LIN {X 0,Y 533.532,Z 613.937,A -85,B 0,C 180,E1 -4225.939,E2 -4225.939} C_VEL
LIN {X 0,Y 532.908,Z 627.148,A -85,B 0,C 180,E1 -4226.975,E2 -4226.975} C_VEL
LIN {X 0,Y 532.504,Z 637.558,A -85,B 0,C 180,E1 -4227.919,E2 -4227.919} C_VEL
LIN {X 0,Y 532.126,Z 646.759,A -85,B 0,C 180,E1 -4228.864,E2 -4228.864} C_VEL
LIN {X 0,Y 531.704,Z 656.519,A -85,B 0,C 180,E1 -4229.999,E2 -4229.999} C_VEL
LIN {X 0,Y 531.313,Z 666.406,A -85,B 0,C 180,E1 -4231.326,E2 -4231.326} C_VEL
LIN {X 0,Y 531.018,Z 676.107,A -85,B 0,C 180,E1 -4232.844,E2 -4232.844} C_VEL
LIN {X 0,Y 530.774,Z 685.128,A -85,B 0,C 180,E1 -4234.556,E2 -4234.556} C_VEL
LIN {X 0,Y 530.628,Z 691.8,A -85,B 0,C 180,E1 -4236.081,E2 -4236.081} C_VEL
LIN {X 0,Y 530.552,Z 697.288,A -85,B 0,C 180,E1 -4237.611,E2 -4237.611} C_VEL
LIN {X 0,Y 530.429,Z 701.704,A -85,B 0,C 180,E1 -4239.148,E2 -4239.148} C_VEL
LIN {X 0,Y 530.423,Z 705.038,A -85,B 0,C 180,E1 -4240.689,E2 -4240.689} C_VEL
LIN {X 0,Y 530.38,Z 707.363,A -85,B 0,C 180,E1 -4242.239,E2 -4242.239} C_VEL
LIN {X 0,Y 530.39,Z 708.671,A -85,B 0,C 180,E1 -4243.798,E2 -4243.798} C_VEL
LIN {X 0,Y 530.314,Z 708.94,A -85,B 0,C 180,E1 -4245.369,E2 -4245.369} C_VEL
LIN {X 0,Y 530.358,Z 708.205,A -85,B 0,C 180,E1 -4246.949,E2 -4246.949} C_VEL
LIN {X 0,Y 530.365,Z 706.395,A -85,B 0,C 180,E1 -4248.543,E2 -4248.543} C_VEL
LIN {X 0,Y 530.391,Z 703.522,A -85,B 0,C 180,E1 -4250.151,E2 -4250.151} C_VEL
LIN {X 0,Y 530.516,Z 698.892,A -85,B 0,C 180,E1 -4251.978,E2 -4251.978} C_VEL
LIN {X 0,Y 530.594,Z 693.091,A -85,B 0,C 180,E1 -4253.684,E2 -4253.684} C_VEL
LIN {X 0,Y 530.727,Z 687.292,A -85,B 0,C 180,E1 -4255.07,E2 -4255.07} C_VEL
LIN {X 0,Y 530.922,Z 680.034,A -85,B 0,C 180,E1 -4256.535,E2 -4256.535} C_VEL
LIN {X 0,Y 531.158,Z 671.391,A -85,B 0,C 180,E1 -4258.015,E2 -4258.015} C_VEL
LIN {X 0,Y 531.539,Z 661.138,A -85,B 0,C 180,E1 -4259.505,E2 -4259.505} C_VEL
LIN {X 0,Y 531.98,Z 650.38,A -85,B 0,C 180,E1 -4260.826,E2 -4260.826} C_VEL
LIN {X 0,Y 532.443,Z 639.033,A -85,B 0,C 180,E1 -4262.027,E2 -4262.027} C_VEL
LIN {X 0,Y 532.896,Z 627.678,A -85,B 0,C 180,E1 -4263.069,E2 -4263.069} C_VEL
LIN {X 0,Y 533.43,Z 615.355,A -85,B 0,C 180,E1 -4264.046,E2 -4264.046} C_VEL
LIN {X 0,Y 534.028,Z 600.641,A -85,B 0,C 180,E1 -4265.037,E2 -4265.037} C_VEL
LIN {X 0,Y 534.612,Z 585.573,A -85,B 0,C 180,E1 -4265.859,E2 -4265.859} C_VEL
LIN {X 0,Y 535.013,Z 571.807,A -85,B 0,C 180,E1 -4266.478,E2 -4266.478} C_VEL
LIN {X 0,Y 535.43,Z 558.758,A -85,B 0,C 180,E1 -4266.948,E2 -4266.948} C_VEL
LIN {X 0,Y 535.723,Z 546.011,A -85,B 0,C 180,E1 -4267.312,E2 -4267.312} C_VEL
LIN {X 0,Y 535.688,Z 538.488,A -85,B 0,C 180,E1 -4267.498,E2 -4267.498} C_VEL
LIN {X 0,Y 530.646,Z 521.655,A -85,B 0,C 180,E1 -4268.016,E2 -4268.016} C_VEL
LIN {X 0,Y 530.688,Z 516.304,A -85,B 0,C 180,E1 -4270.986,E2 -4270.986} C_VEL
LIN {X 0,Y 530.788,Z 512.053,A -85,B 0,C 180,E1 -4273.511,E2 -4273.511} C_VEL
LIN {X 0,Y 530.883,Z 506.871,A -85,B 0,C 180,E1 -4276.496,E2 -4276.496} C_VEL
LIN {X 0,Y 530.93,Z 502.507,A -85,B 0,C 180,E1 -4278.981,E2 -4278.981} C_VEL
LIN {X 0,Y 530.941,Z 497.816,A -85,B 0,C 180,E1 -4281.527,E2 -4281.527} C_VEL
LIN {X 0,Y 531.038,Z 492.653,A -85,B 0,C 180,E1 -4284.288,E2 -4284.288} C_VEL
LIN {X 0,Y 530.968,Z 492.661,A -85,B 0,C 180,E1 -4287.133,E2 -4287.133} C_VEL
LIN {X 0,Y 530.979,Z 492.659,A -85,B 0,C 180,E1 -4289.803,E2 -4289.803} C_VEL
LIN {X 0,Y 531.01,Z 492.655,A -85,B 0,C 180,E1 -4292.465,E2 -4292.465} C_VEL
LIN {X 0,Y 531.007,Z 492.656,A -85,B 0,C 180,E1 -4294.942,E2 -4294.942} C_VEL
LIN {X 0,Y 530.983,Z 492.658,A -85,B 0,C 180,E1 -4297.893,E2 -4297.893} C_VEL
LIN {X 0,Y 530.989,Z 492.655,A -85,B 0,C 180,E1 -4300.677,E2 -4300.677} C_VEL
LIN {X 0,Y 530.984,Z 492.658,A -85,B 0,C 180,E1 -4303.071,E2 -4303.071} C_VEL
LIN {X 0,Y 531.009,Z 492.654,A -85,B 0,C 180,E1 -4305.435,E2 -4305.435} C_VEL
LIN {X 0,Y 531.037,Z 492.65,A -85,B 0,C 180,E1 -4308.549,E2 -4308.549} C_VEL
LIN {X 0,Y 531.051,Z 492.646,A -85,B 0,C 180,E1 -4311.629,E2 -4311.629} C_VEL
LIN {X 0,Y 531.137,Z 492.636,A -85,B 0,C 180,E1 -4314.685,E2 -4314.685} C_VEL
LIN {X 0,Y 531.134,Z 492.639,A -85,B 0,C 180,E1 -4317.725,E2 -4317.725} C_VEL
LIN {X 0,Y 531.147,Z 492.638,A -85,B 0,C 180,E1 -4320.758,E2 -4320.758} C_VEL
LIN {X 0,Y 531.101,Z 492.641,A -85,B 0,C 180,E1 -4323.034,E2 -4323.034} C_VEL
LIN {X 0,Y 531.074,Z 492.645,A -85,B 0,C 180,E1 -4326.077,E2 -4326.077} C_VEL
LIN {X 0,Y 531.026,Z 492.65,A -85,B 0,C 180,E1 -4329.138,E2 -4329.138} C_VEL
LIN {X 0,Y 531.03,Z 492.647,A -85,B 0,C 180,E1 -4332.225,E2 -4332.225} C_VEL
LIN {X 0,Y 530.985,Z 492.656,A -85,B 0,C 180,E1 -4335.35,E2 -4335.35} C_VEL
LIN {X 0,Y 531.005,Z 492.639,A -85,B 0,C 180,E1 -4337.722,E2 -4337.722} C_VEL
LIN {X 0,Y 530.994,Z 492.657,A -85,B 0,C 180,E1 -4340.938,E2 -4340.938} C_VEL
LIN {X 0,Y 530.997,Z 492.644,A -85,B 0,C 180,E1 -4344.045,E2 -4344.045} C_VEL
LIN {X 0,Y 531.002,Z 492.655,A -85,B 0,C 180,E1 -4346.743,E2 -4346.743} C_VEL
LIN {X 0,Y 530.99,Z 492.658,A -85,B 0,C 180,E1 -4349.322,E2 -4349.322} C_VEL
LIN {X 0,Y 530.97,Z 492.66,A -85,B 0,C 180,E1 -4352.104,E2 -4352.104} C_VEL
LIN {X 0,Y 530.982,Z 492.657,A -85,B 0,C 180,E1 -4354.855,E2 -4354.855} C_VEL
LIN {X 0,Y 530.964,Z 492.66,A -85,B 0,C 180,E1 -4357.507,E2 -4357.507} C_VEL
LIN {X 0,Y 531.019,Z 492.652,A -85,B 0,C 180,E1 -4360.429,E2 -4360.429} C_VEL
LIN {X 0,Y 530.957,Z 492.661,A -85,B 0,C 180,E1 -4363.495,E2 -4363.495} C_VEL
LIN {X 0,Y 531.009,Z 492.819,A -85,B 0,C 180,E1 -4366.402,E2 -4366.402} C_VEL
LIN {X 0,Y 532.868,Z 501.243,A -85,B 0,C 180,E1 -4368.744,E2 -4368.744} C_VEL
LIN {X 0,Y 533.677,Z 505.22,A -85,B 0,C 180,E1 -4369.815,E2 -4369.815} C_VEL
LIN {X 0,Y 533.689,Z 513.013,A -85,B 0,C 180,E1 -4371.764,E2 -4371.764} C_VEL
LIN {X 0,Y 533.387,Z 525.433,A -85,B 0,C 180,E1 -4374.777,E2 -4374.777} C_VEL
LIN {X 0,Y 532.901,Z 537.907,A -85,B 0,C 180,E1 -4377.86,E2 -4377.86} C_VEL
LIN {X 0,Y 532.51,Z 550.04,A -85,B 0,C 180,E1 -4380.771,E2 -4380.771} C_VEL
LIN {X 0,Y 532.194,Z 560.938,A -85,B 0,C 180,E1 -4383.322,E2 -4383.322} C_VEL
LIN {X 0,Y 531.825,Z 573.652,A -85,B 0,C 180,E1 -4386.232,E2 -4386.232} C_VEL
LIN {X 0,Y 531.761,Z 577.116,A -85,B 0,C 180,E1 -4387.016,E2 -4387.016} C_VEL
LIN {X 0,Y 535.893,Z 592.599,A -85,B 0,C 180,E1 -4387.446,E2 -4387.446} C_VEL
LIN {X 0,Y 535.686,Z 608.888,A -85,B 0,C 180,E1 -4387.805,E2 -4387.805} C_VEL
LIN {X 0,Y 535.309,Z 624.847,A -85,B 0,C 180,E1 -4388.3,E2 -4388.3} C_VEL
LIN {X 0,Y 534.788,Z 640.031,A -85,B 0,C 180,E1 -4388.916,E2 -4388.916} C_VEL
LIN {X 0,Y 534.26,Z 655.297,A -85,B 0,C 180,E1 -4389.7,E2 -4389.7} C_VEL
LIN {X 0,Y 533.646,Z 670.869,A -85,B 0,C 180,E1 -4390.678,E2 -4390.678} C_VEL
LIN {X 0,Y 533.025,Z 685.379,A -85,B 0,C 180,E1 -4391.779,E2 -4391.779} C_VEL
LIN {X 0,Y 532.488,Z 698.13,A -85,B 0,C 180,E1 -4392.924,E2 -4392.924} C_VEL
LIN {X 0,Y 532.031,Z 709.292,A -85,B 0,C 180,E1 -4394.093,E2 -4394.093} C_VEL
LIN {X 0,Y 531.635,Z 720.431,A -85,B 0,C 180,E1 -4395.454,E2 -4395.454} C_VEL
LIN {X 0,Y 531.191,Z 731.218,A -85,B 0,C 180,E1 -4397.003,E2 -4397.003} C_VEL
LIN {X 0,Y 530.965,Z 740.269,A -85,B 0,C 180,E1 -4398.549,E2 -4398.549} C_VEL
LIN {X 0,Y 530.696,Z 747.861,A -85,B 0,C 180,E1 -4400.088,E2 -4400.088} C_VEL
LIN {X 0,Y 530.568,Z 755.47,A -85,B 0,C 180,E1 -4402.006,E2 -4402.006} C_VEL
LIN {X 0,Y 530.494,Z 761.25,A -85,B 0,C 180,E1 -4403.917,E2 -4403.917} C_VEL
LIN {X 0,Y 530.403,Z 764.638,A -85,B 0,C 180,E1 -4405.441,E2 -4405.441} C_VEL
LIN {X 0,Y 530.444,Z 767.09,A -85,B 0,C 180,E1 -4406.963,E2 -4406.963} C_VEL
LIN {X 0,Y 530.357,Z 768.48,A -85,B 0,C 180,E1 -4408.482,E2 -4408.482} C_VEL
LIN {X 0,Y 530.338,Z 769,A -85,B 0,C 180,E1 -4410.001,E2 -4410.001} C_VEL
LIN {X 0,Y 530.357,Z 768.479,A -85,B 0,C 180,E1 -4411.519,E2 -4411.519} C_VEL
LIN {X 0,Y 530.444,Z 767.087,A -85,B 0,C 180,E1 -4413.039,E2 -4413.039} C_VEL
LIN {X 0,Y 530.404,Z 764.635,A -85,B 0,C 180,E1 -4414.561,E2 -4414.561} C_VEL
LIN {X 0,Y 530.494,Z 761.247,A -85,B 0,C 180,E1 -4416.085,E2 -4416.085} C_VEL
LIN {X 0,Y 530.57,Z 755.465,A -85,B 0,C 180,E1 -4417.996,E2 -4417.996} C_VEL
LIN {X 0,Y 530.697,Z 747.853,A -85,B 0,C 180,E1 -4419.914,E2 -4419.914} C_VEL
LIN {X 0,Y 531.001,Z 739.244,A -85,B 0,C 180,E1 -4421.646,E2 -4421.646} C_VEL
LIN {X 0,Y 531.229,Z 729.97,A -85,B 0,C 180,E1 -4423.193,E2 -4423.193} C_VEL
LIN {X 0,Y 531.68,Z 719.216,A -85,B 0,C 180,E1 -4424.704,E2 -4424.704} C_VEL
LIN {X 0,Y 532.103,Z 707.5,A -85,B 0,C 180,E1 -4426.104,E2 -4426.104} C_VEL
LIN {X 0,Y 532.631,Z 695.034,A -85,B 0,C 180,E1 -4427.37,E2 -4427.37} C_VEL
LIN {X 0,Y 533.201,Z 681.455,A -85,B 0,C 180,E1 -4428.542,E2 -4428.542} C_VEL
LIN {X 0,Y 533.812,Z 666.56,A -85,B 0,C 180,E1 -4429.617,E2 -4429.617} C_VEL
LIN {X 0,Y 534.389,Z 651.742,A -85,B 0,C 180,E1 -4430.498,E2 -4430.498} C_VEL
LIN {X 0,Y 534.889,Z 637.688,A -85,B 0,C 180,E1 -4431.185,E2 -4431.185} C_VEL
LIN {X 0,Y 535.393,Z 622.424,A -85,B 0,C 180,E1 -4431.787,E2 -4431.787} C_VEL
LIN {X 0,Y 535.698,Z 606.492,A -85,B 0,C 180,E1 -4432.261,E2 -4432.261} C_VEL
LIN {X 0,Y 535.767,Z 592.182,A -85,B 0,C 180,E1 -4432.567,E2 -4432.567} C_VEL
LIN {X 0,Y 531.754,Z 577.091,A -85,B 0,C 180,E1 -4432.99,E2 -4432.99} C_VEL
LIN {X 0,Y 532.176,Z 562.417,A -85,B 0,C 180,E1 -4436.335,E2 -4436.335} C_VEL
LIN {X 0,Y 532.517,Z 550.032,A -85,B 0,C 180,E1 -4439.23,E2 -4439.23} C_VEL
LIN {X 0,Y 532.907,Z 537.9,A -85,B 0,C 180,E1 -4442.142,E2 -4442.142} C_VEL
LIN {X 0,Y 533.437,Z 524.602,A -85,B 0,C 180,E1 -4445.43,E2 -4445.43} C_VEL
LIN {X 0,Y 533.404,Z 512.664,A -85,B 0,C 180,E1 -4447.973,E2 -4447.973} C_VEL
LIN {X 0,Y 533.144,Z 503.532,A -85,B 0,C 180,E1 -4449.886,E2 -4449.886} C_VEL
LIN {X 0,Y 530.993,Z 492.658,A -85,B 0,C 180,E1 -4452.38,E2 -4452.38} C_VEL
LIN {X 0,Y 530.989,Z 492.654,A -85,B 0,C 180,E1 -4455.621,E2 -4455.621} C_VEL
LIN {X 0,Y 530.997,Z 492.658,A -85,B 0,C 180,E1 -4458.565,E2 -4458.565} C_VEL
LIN {X 0,Y 530.96,Z 492.657,A -85,B 0,C 180,E1 -4461.53,E2 -4461.53} C_VEL
LIN {X 0,Y 530.978,Z 492.661,A -85,B 0,C 180,E1 -4464.382,E2 -4464.382} C_VEL
LIN {X 0,Y 530.971,Z 492.656,A -85,B 0,C 180,E1 -4467.134,E2 -4467.134} C_VEL
LIN {X 0,Y 530.971,Z 492.659,A -85,B 0,C 180,E1 -4469.803,E2 -4469.803} C_VEL
LIN {X 0,Y 531.018,Z 492.653,A -85,B 0,C 180,E1 -4472.467,E2 -4472.467} C_VEL
LIN {X 0,Y 531.008,Z 492.651,A -85,B 0,C 180,E1 -4474.943,E2 -4474.943} C_VEL
LIN {X 0,Y 530.972,Z 492.658,A -85,B 0,C 180,E1 -4477.265,E2 -4477.265} C_VEL
LIN {X 0,Y 532.385,Z 496.563,A -85,B 0,C 180,E1 -4477.408,E2 -4477.408} C_VEL
LIN {X 0,Y 535.775,Z 504.819,A -85,B 0,C 180,E1 -4477.744,E2 -4477.744} C_VEL
LIN {X 0,Y 535.408,Z 520.411,A -85,B 0,C 180,E1 -4478.188,E2 -4478.188} C_VEL
LIN {X 0,Y 534.945,Z 536.534,A -85,B 0,C 180,E1 -4478.808,E2 -4478.808} C_VEL
LIN {X 0,Y 534.336,Z 552.771,A -85,B 0,C 180,E1 -4479.602,E2 -4479.602} C_VEL
LIN {X 0,Y 533.789,Z 567.376,A -85,B 0,C 180,E1 -4480.483,E2 -4480.483} C_VEL
LIN {X 0,Y 533.198,Z 582.144,A -85,B 0,C 180,E1 -4481.559,E2 -4481.559} C_VEL
LIN {X 0,Y 532.638,Z 595.622,A -85,B 0,C 180,E1 -4482.73,E2 -4482.73} C_VEL
LIN {X 0,Y 532.104,Z 607.116,A -85,B 0,C 180,E1 -4483.897,E2 -4483.897} C_VEL
LIN {X 0,Y 531.704,Z 618.906,A -85,B 0,C 180,E1 -4485.297,E2 -4485.297} C_VEL
LIN {X 0,Y 531.229,Z 629.714,A -85,B 0,C 180,E1 -4486.808,E2 -4486.808} C_VEL
LIN {X 0,Y 531.003,Z 638.994,A -85,B 0,C 180,E1 -4488.355,E2 -4488.355} C_VEL
LIN {X 0,Y 530.699,Z 647.635,A -85,B 0,C 180,E1 -4490.087,E2 -4490.087} C_VEL
LIN {X 0,Y 530.604,Z 653.896,A -85,B 0,C 180,E1 -4491.623,E2 -4491.623} C_VEL
LIN {X 0,Y 530.549,Z 658.995,A -85,B 0,C 180,E1 -4493.153,E2 -4493.153} C_VEL
LIN {X 0,Y 530.472,Z 662.97,A -85,B 0,C 180,E1 -4494.679,E2 -4494.679} C_VEL
LIN {X 0,Y 530.478,Z 665.916,A -85,B 0,C 180,E1 -4496.202,E2 -4496.202} C_VEL
LIN {X 0,Y 530.403,Z 667.872,A -85,B 0,C 180,E1 -4497.722,E2 -4497.722} C_VEL
LIN {X 0,Y 530.342,Z 668.857,A -85,B 0,C 180,E1 -4499.241,E2 -4499.241} C_VEL
LIN {X 0,Y 530.341,Z 668.874,A -85,B 0,C 180,E1 -4500.76,E2 -4500.76} C_VEL
LIN {X 0,Y 530.403,Z 667.951,A -85,B 0,C 180,E1 -4502.279,E2 -4502.279} C_VEL
LIN {X 0,Y 530.48,Z 666.057,A -85,B 0,C 180,E1 -4503.799,E2 -4503.799} C_VEL
LIN {X 0,Y 530.472,Z 663.168,A -85,B 0,C 180,E1 -4505.322,E2 -4505.322} C_VEL
LIN {X 0,Y 530.55,Z 659.27,A -85,B 0,C 180,E1 -4506.847,E2 -4506.847} C_VEL
LIN {X 0,Y 530.604,Z 654.24,A -85,B 0,C 180,E1 -4508.378,E2 -4508.378} C_VEL
LIN {X 0,Y 530.695,Z 648.056,A -85,B 0,C 180,E1 -4509.914,E2 -4509.914} C_VEL
LIN {X 0,Y 530.977,Z 639.556,A -85,B 0,C 180,E1 -4511.632,E2 -4511.632} C_VEL
LIN {X 0,Y 531.226,Z 630.266,A -85,B 0,C 180,E1 -4513.192,E2 -4513.192} C_VEL
LIN {X 0,Y 531.675,Z 619.59,A -85,B 0,C 180,E1 -4514.704,E2 -4514.704} C_VEL
LIN {X 0,Y 532.077,Z 607.953,A -85,B 0,C 180,E1 -4516.104,E2 -4516.104} C_VEL
LIN {X 0,Y 532.598,Z 595.538,A -85,B 0,C 180,E1 -4517.371,E2 -4517.371} C_VEL
LIN {X 0,Y 533.19,Z 582,A -85,B 0,C 180,E1 -4518.542,E2 -4518.542} C_VEL
LIN {X 0,Y 533.804,Z 567.184,A -85,B 0,C 180,E1 -4519.617,E2 -4519.617} C_VEL
LIN {X 0,Y 534.384,Z 552.56,A -85,B 0,C 180,E1 -4520.498,E2 -4520.498} C_VEL
LIN {X 0,Y 534.932,Z 537.448,A -85,B 0,C 180,E1 -4521.243,E2 -4521.243} C_VEL
LIN {X 0,Y 535.376,Z 520.293,A -85,B 0,C 180,E1 -4521.901,E2 -4521.901} C_VEL
LIN {X 0,Y 535.732,Z 506.697,A -85,B 0,C 180,E1 -4522.294,E2 -4522.294} C_VEL
LIN {X 0,Y 535.554,Z 504.031,A -85,B 0,C 180,E1 -4522.369,E2 -4522.369} C_VEL
LIN {X 0,Y 531.057,Z 493.147,A -85,B 0,C 180,E1 -4522.801,E2 -4522.801} C_VEL
LIN {X 0,Y 530.977,Z 492.659,A -85,B 0,C 180,E1 -4522.834,E2 -4522.834} C_VEL
LIN {X 0,Y 531.017,Z 492.654,A -85,B 0,C 180,E1 -4525.897,E2 -4525.897} C_VEL
LIN {X 0,Y 531,Z 492.654,A -85,B 0,C 180,E1 -4528.456,E2 -4528.456} C_VEL
LIN {X 0,Y 530.954,Z 492.659,A -85,B 0,C 180,E1 -4531.219,E2 -4531.219} C_VEL
LIN {X 0,Y 530.994,Z 492.654,A -85,B 0,C 180,E1 -4533.773,E2 -4533.773} C_VEL
LIN {X 0,Y 530.99,Z 492.657,A -85,B 0,C 180,E1 -4534.524,E2 -4534.524} C_VEL
LIN {X 0,Y 530.348,Z 492.742,A -85,B 0,C 180,E1 -4535.157,E2 -4535.157} C_VEL
LIN {X 0,Y 527.476,Z 493.102,A -85,B 0,C 180,E1 -4536.184,E2 -4536.184} C_VEL
LIN {X 0,Y 525.035,Z 493.403,A -85,B 0,C 180,E1 -4537.011,E2 -4537.011} C_VEL
LIN {X 0,Y 523.993,Z 493.529,A -85,B 0,C 180,E1 -4537.65,E2 -4537.65} C_VEL
LIN {X 0,Y 523.913,Z 493.537,A -85,B 0,C 180,E1 -4537.866,E2 -4537.866} C_VEL
LIN {X 0,Y 523.943,Z 493.533,A -85,B 0,C 180,E1 -4541.092,E2 -4541.092} C_VEL
LIN {X 0,Y 523.936,Z 493.534,A -85,B 0,C 180,E1 -4544.229,E2 -4544.229} C_VEL
LIN {X 0,Y 523.927,Z 493.534,A -85,B 0,C 180,E1 -4546.833,E2 -4546.833} C_VEL
LIN {X 0,Y 523.95,Z 493.536,A -85,B 0,C 180,E1 -4548.908,E2 -4548.908} C_VEL
LIN {X 0,Y 523.921,Z 493.539,A -85,B 0,C 180,E1 -4551.898,E2 -4551.898} C_VEL
LIN {X 0,Y 523.93,Z 493.537,A -85,B 0,C 180,E1 -4554.911,E2 -4554.911} C_VEL
LIN {X 0,Y 523.941,Z 493.538,A -85,B 0,C 180,E1 -4557.68,E2 -4557.68} C_VEL
LIN {X 0,Y 523.96,Z 493.534,A -85,B 0,C 180,E1 -4560.676,E2 -4560.676} C_VEL
LIN {X 0,Y 523.98,Z 493.53,A -85,B 0,C 180,E1 -4563.728,E2 -4563.728} C_VEL
LIN {X 0,Y 524.052,Z 493.703,A -85,B 0,C 180,E1 -4565.776,E2 -4565.776} C_VEL
LIN {X 0,Y 523.943,Z 499.278,A -85,B 0,C 180,E1 -4568.766,E2 -4568.766} C_VEL
LIN {X 0,Y 523.917,Z 503.685,A -85,B 0,C 180,E1 -4571.219,E2 -4571.219} C_VEL
LIN {X 0,Y 523.847,Z 507.921,A -85,B 0,C 180,E1 -4573.635,E2 -4573.635} C_VEL
LIN {X 0,Y 523.803,Z 512.025,A -85,B 0,C 180,E1 -4576.024,E2 -4576.024} C_VEL
LIN {X 0,Y 523.75,Z 517.352,A -85,B 0,C 180,E1 -4579.171,E2 -4579.171} C_VEL
LIN {X 0,Y 523.652,Z 521.772,A -85,B 0,C 180,E1 -4581.759,E2 -4581.759} C_VEL
LIN {X 0,Y 526.868,Z 532.431,A -85,B 0,C 180,E1 -4582.085,E2 -4582.085} C_VEL
LIN {X 0,Y 529.265,Z 540.268,A -85,B 0,C 180,E1 -4582.345,E2 -4582.345} C_VEL
LIN {X 0,Y 528.905,Z 556.103,A -85,B 0,C 180,E1 -4582.769,E2 -4582.769} C_VEL
LIN {X 0,Y 528.485,Z 569.08,A -85,B 0,C 180,E1 -4583.221,E2 -4583.221} C_VEL
LIN {X 0,Y 527.992,Z 582.219,A -85,B 0,C 180,E1 -4583.791,E2 -4583.791} C_VEL
LIN {X 0,Y 527.526,Z 594.897,A -85,B 0,C 180,E1 -4584.456,E2 -4584.456} C_VEL
LIN {X 0,Y 527.031,Z 607.205,A -85,B 0,C 180,E1 -4585.218,E2 -4585.218} C_VEL
LIN {X 0,Y 526.495,Z 619.1,A -85,B 0,C 180,E1 -4586.076,E2 -4586.076} C_VEL
LIN {X 0,Y 525.876,Z 632.738,A -85,B 0,C 180,E1 -4587.222,E2 -4587.222} C_VEL
LIN {X 0,Y 525.282,Z 645.152,A -85,B 0,C 180,E1 -4588.466,E2 -4588.466} C_VEL
LIN {X 0,Y 524.848,Z 655.086,A -85,B 0,C 180,E1 -4589.616,E2 -4589.616} C_VEL
LIN {X 0,Y 524.397,Z 663.818,A -85,B 0,C 180,E1 -4590.767,E2 -4590.767} C_VEL
LIN {X 0,Y 524.127,Z 672.686,A -85,B 0,C 180,E1 -4592.112,E2 -4592.112} C_VEL
LIN {X 0,Y 523.808,Z 680.366,A -85,B 0,C 180,E1 -4593.461,E2 -4593.461} C_VEL
LIN {X 0,Y 523.647,Z 687.846,A -85,B 0,C 180,E1 -4595.004,E2 -4595.004} C_VEL
LIN {X 0,Y 523.525,Z 694.184,A -85,B 0,C 180,E1 -4596.581,E2 -4596.581} C_VEL
LIN {X 0,Y 523.47,Z 699.124,A -85,B 0,C 180,E1 -4598.103,E2 -4598.103} C_VEL
LIN {X 0,Y 523.323,Z 702.221,A -85,B 0,C 180,E1 -4599.273,E2 -4599.273} C_VEL
LIN {X 0,Y 523.35,Z 705.419,A -85,B 0,C 180,E1 -4600.835,E2 -4600.835} C_VEL
LIN {X 0,Y 523.28,Z 707.574,A -85,B 0,C 180,E1 -4602.408,E2 -4602.408} C_VEL
LIN {X 0,Y 523.28,Z 708.734,A -85,B 0,C 180,E1 -4603.989,E2 -4603.989} C_VEL
LIN {X 0,Y 523.221,Z 708.883,A -85,B 0,C 180,E1 -4605.583,E2 -4605.583} C_VEL
LIN {X 0,Y 523.287,Z 708.018,A -85,B 0,C 180,E1 -4607.185,E2 -4607.185} C_VEL
LIN {X 0,Y 523.26,Z 706.084,A -85,B 0,C 180,E1 -4608.804,E2 -4608.804} C_VEL
LIN {X 0,Y 523.312,Z 703.078,A -85,B 0,C 180,E1 -4610.436,E2 -4610.436} C_VEL
LIN {X 0,Y 523.435,Z 698.778,A -85,B 0,C 180,E1 -4612.112,E2 -4612.112} C_VEL
LIN {X 0,Y 523.513,Z 693.295,A -85,B 0,C 180,E1 -4613.748,E2 -4613.748} C_VEL
LIN {X 0,Y 523.646,Z 688.204,A -85,B 0,C 180,E1 -4615.008,E2 -4615.008} C_VEL
LIN {X 0,Y 523.853,Z 681.095,A -85,B 0,C 180,E1 -4616.491,E2 -4616.491} C_VEL
LIN {X 0,Y 524.111,Z 672.617,A -85,B 0,C 180,E1 -4617.989,E2 -4617.989} C_VEL
LIN {X 0,Y 524.434,Z 664.633,A -85,B 0,C 180,E1 -4619.204,E2 -4619.204} C_VEL
LIN {X 0,Y 524.876,Z 654.228,A -85,B 0,C 180,E1 -4620.583,E2 -4620.583} C_VEL
LIN {X 0,Y 525.515,Z 640.48,A -85,B 0,C 180,E1 -4622.112,E2 -4622.112} C_VEL
LIN {X 0,Y 526.02,Z 628.785,A -85,B 0,C 180,E1 -4623.214,E2 -4623.214} C_VEL
LIN {X 0,Y 526.559,Z 617.252,A -85,B 0,C 180,E1 -4624.155,E2 -4624.155} C_VEL
LIN {X 0,Y 527.089,Z 605.541,A -85,B 0,C 180,E1 -4624.982,E2 -4624.982} C_VEL
LIN {X 0,Y 527.674,Z 592.213,A -85,B 0,C 180,E1 -4625.785,E2 -4625.785} C_VEL
LIN {X 0,Y 528.279,Z 575.89,A -85,B 0,C 180,E1 -4626.594,E2 -4626.594} C_VEL
LIN {X 0,Y 528.754,Z 560.414,A -85,B 0,C 180,E1 -4627.183,E2 -4627.183} C_VEL
LIN {X 0,Y 529.096,Z 547.881,A -85,B 0,C 180,E1 -4627.557,E2 -4627.557} C_VEL
LIN {X 0,Y 529.112,Z 540.073,A -85,B 0,C 180,E1 -4627.757,E2 -4627.757} C_VEL
LIN {X 0,Y 523.561,Z 521.696,A -85,B 0,C 180,E1 -4628.337,E2 -4628.337} C_VEL
LIN {X 0,Y 523.685,Z 516.83,A -85,B 0,C 180,E1 -4631.276,E2 -4631.276} C_VEL
LIN {X 0,Y 523.768,Z 512.939,A -85,B 0,C 180,E1 -4633.565,E2 -4633.565} C_VEL
LIN {X 0,Y 523.871,Z 508.037,A -85,B 0,C 180,E1 -4636.42,E2 -4636.42} C_VEL
LIN {X 0,Y 523.89,Z 503.577,A -85,B 0,C 180,E1 -4638.902,E2 -4638.902} C_VEL
LIN {X 0,Y 523.943,Z 499.638,A -85,B 0,C 180,E1 -4641.075,E2 -4641.075} C_VEL
LIN {X 0,Y 523.999,Z 493.53,A -85,B 0,C 180,E1 -4644.307,E2 -4644.307} C_VEL
LIN {X 0,Y 523.933,Z 493.537,A -85,B 0,C 180,E1 -4647.55,E2 -4647.55} C_VEL
LIN {X 0,Y 523.962,Z 493.534,A -85,B 0,C 180,E1 -4650.672,E2 -4650.672} C_VEL
LIN {X 0,Y 523.97,Z 493.533,A -85,B 0,C 180,E1 -4653.728,E2 -4653.728} C_VEL
LIN {X 0,Y 523.942,Z 493.536,A -85,B 0,C 180,E1 -4656.271,E2 -4656.271} C_VEL
LIN {X 0,Y 523.944,Z 493.536,A -85,B 0,C 180,E1 -4658.766,E2 -4658.766} C_VEL
LIN {X 0,Y 523.946,Z 493.532,A -85,B 0,C 180,E1 -4661.22,E2 -4661.22} C_VEL
LIN {X 0,Y 523.931,Z 493.533,A -85,B 0,C 180,E1 -4663.638,E2 -4663.638} C_VEL
LIN {X 0,Y 523.932,Z 493.534,A -85,B 0,C 180,E1 -4666.027,E2 -4666.027} C_VEL
LIN {X 0,Y 524.001,Z 493.528,A -85,B 0,C 180,E1 -4668.394,E2 -4668.394} C_VEL
LIN {X 0,Y 523.999,Z 493.525,A -85,B 0,C 180,E1 -4671.516,E2 -4671.516} C_VEL
LIN {X 0,Y 524.095,Z 493.513,A -85,B 0,C 180,E1 -4674.613,E2 -4674.613} C_VEL
LIN {X 0,Y 524.106,Z 493.514,A -85,B 0,C 180,E1 -4677.694,E2 -4677.694} C_VEL
LIN {X 0,Y 524.117,Z 493.513,A -85,B 0,C 180,E1 -4680.768,E2 -4680.768} C_VEL
LIN {X 0,Y 524.067,Z 493.517,A -85,B 0,C 180,E1 -4683.075,E2 -4683.075} C_VEL
LIN {X 0,Y 524.036,Z 493.522,A -85,B 0,C 180,E1 -4686.159,E2 -4686.159} C_VEL
LIN {X 0,Y 523.994,Z 493.525,A -85,B 0,C 180,E1 -4689.262,E2 -4689.262} C_VEL
LIN {X 0,Y 524.013,Z 493.523,A -85,B 0,C 180,E1 -4691.751,E2 -4691.751} C_VEL
LIN {X 0,Y 523.981,Z 493.527,A -85,B 0,C 180,E1 -4695.052,E2 -4695.052} C_VEL
LIN {X 0,Y 523.953,Z 493.517,A -85,B 0,C 180,E1 -4697.969,E2 -4697.969} C_VEL
LIN {X 0,Y 523.962,Z 493.53,A -85,B 0,C 180,E1 -4700.41,E2 -4700.41} C_VEL
LIN {X 0,Y 523.933,Z 493.53,A -85,B 0,C 180,E1 -4702.892,E2 -4702.892} C_VEL
LIN {X 0,Y 523.975,Z 493.524,A -85,B 0,C 180,E1 -4706.021,E2 -4706.021} C_VEL
LIN {X 0,Y 523.94,Z 493.534,A -85,B 0,C 180,E1 -4708.874,E2 -4708.874} C_VEL
LIN {X 0,Y 523.923,Z 493.536,A -85,B 0,C 180,E1 -4711.544,E2 -4711.544} C_VEL
LIN {X 0,Y 523.936,Z 493.534,A -85,B 0,C 180,E1 -4714.29,E2 -4714.29} C_VEL
LIN {X 0,Y 523.908,Z 493.538,A -85,B 0,C 180,E1 -4717.132,E2 -4717.132} C_VEL
LIN {X 0,Y 523.984,Z 493.53,A -85,B 0,C 180,E1 -4720.138,E2 -4720.138} C_VEL
LIN {X 0,Y 523.916,Z 493.539,A -85,B 0,C 180,E1 -4723.167,E2 -4723.167} C_VEL
LIN {X 0,Y 523.957,Z 493.652,A -85,B 0,C 180,E1 -4726.015,E2 -4726.015} C_VEL
LIN {X 0,Y 526.122,Z 503.486,A -85,B 0,C 180,E1 -4728.799,E2 -4728.799} C_VEL
LIN {X 0,Y 526.86,Z 507.39,A -85,B 0,C 180,E1 -4729.859,E2 -4729.859} C_VEL
LIN {X 0,Y 526.789,Z 515.574,A -85,B 0,C 180,E1 -4731.918,E2 -4731.918} C_VEL
LIN {X 0,Y 526.55,Z 526.155,A -85,B 0,C 180,E1 -4734.506,E2 -4734.506} C_VEL
LIN {X 0,Y 526.041,Z 539.142,A -85,B 0,C 180,E1 -4737.698,E2 -4737.698} C_VEL
LIN {X 0,Y 525.587,Z 551.856,A -85,B 0,C 180,E1 -4740.788,E2 -4740.788} C_VEL
LIN {X 0,Y 525.218,Z 564.183,A -85,B 0,C 180,E1 -4743.706,E2 -4743.706} C_VEL
LIN {X 0,Y 524.833,Z 577.258,A -85,B 0,C 180,E1 -4746.703,E2 -4746.703} C_VEL
LIN {X 0,Y 529.307,Z 593.893,A -85,B 0,C 180,E1 -4747.172,E2 -4747.172} C_VEL
LIN {X 0,Y 529.101,Z 609.808,A -85,B 0,C 180,E1 -4747.539,E2 -4747.539} C_VEL
LIN {X 0,Y 528.63,Z 626.205,A -85,B 0,C 180,E1 -4748.065,E2 -4748.065} C_VEL
LIN {X 0,Y 528.119,Z 640.851,A -85,B 0,C 180,E1 -4748.674,E2 -4748.674} C_VEL
LIN {X 0,Y 527.482,Z 657.047,A -85,B 0,C 180,E1 -4749.529,E2 -4749.529} C_VEL
LIN {X 0,Y 526.844,Z 672.282,A -85,B 0,C 180,E1 -4750.52,E2 -4750.52} C_VEL
LIN {X 0,Y 526.207,Z 684.858,A -85,B 0,C 180,E1 -4751.49,E2 -4751.49} C_VEL
LIN {X 0,Y 525.626,Z 698.13,A -85,B 0,C 180,E1 -4752.694,E2 -4752.694} C_VEL
LIN {X 0,Y 525.122,Z 709.293,A -85,B 0,C 180,E1 -4753.878,E2 -4753.878} C_VEL
LIN {X 0,Y 524.685,Z 720.43,A -85,B 0,C 180,E1 -4755.257,E2 -4755.257} C_VEL
LIN {X 0,Y 524.175,Z 731.218,A -85,B 0,C 180,E1 -4756.826,E2 -4756.826} C_VEL
LIN {X 0,Y 523.932,Z 740.27,A -85,B 0,C 180,E1 -4758.393,E2 -4758.393} C_VEL
LIN {X 0,Y 523.657,Z 747.86,A -85,B 0,C 180,E1 -4759.953,E2 -4759.953} C_VEL
LIN {X 0,Y 523.503,Z 755.469,A -85,B 0,C 180,E1 -4761.897,E2 -4761.897} C_VEL
LIN {X 0,Y 523.448,Z 760.296,A -85,B 0,C 180,E1 -4763.487,E2 -4763.487} C_VEL
LIN {X 0,Y 523.396,Z 763.061,A -85,B 0,C 180,E1 -4764.607,E2 -4764.607} C_VEL
LIN {X 0,Y 523.398,Z 765.982,A -85,B 0,C 180,E1 -4766.151,E2 -4766.151} C_VEL
LIN {X 0,Y 523.328,Z 767.894,A -85,B 0,C 180,E1 -4767.692,E2 -4767.692} C_VEL
LIN {X 0,Y 523.247,Z 768.849,A -85,B 0,C 180,E1 -4769.231,E2 -4769.231} C_VEL
LIN {X 0,Y 523.247,Z 768.849,A -85,B 0,C 180,E1 -4770.77,E2 -4770.77} C_VEL
LIN {X 0,Y 523.328,Z 767.892,A -85,B 0,C 180,E1 -4772.31,E2 -4772.31} C_VEL
LIN {X 0,Y 523.398,Z 765.979,A -85,B 0,C 180,E1 -4773.85,E2 -4773.85} C_VEL
LIN {X 0,Y 523.397,Z 763.058,A -85,B 0,C 180,E1 -4775.394,E2 -4775.394} C_VEL
LIN {X 0,Y 523.478,Z 759.122,A -85,B 0,C 180,E1 -4776.941,E2 -4776.941} C_VEL
LIN {X 0,Y 523.525,Z 754.047,A -85,B 0,C 180,E1 -4778.493,E2 -4778.493} C_VEL
LIN {X 0,Y 523.658,Z 747.853,A -85,B 0,C 180,E1 -4780.049,E2 -4780.049} C_VEL
LIN {X 0,Y 523.957,Z 739.703,A -85,B 0,C 180,E1 -4781.716,E2 -4781.716} C_VEL
LIN {X 0,Y 524.177,Z 731.208,A -85,B 0,C 180,E1 -4783.176,E2 -4783.176} C_VEL
LIN {X 0,Y 524.687,Z 720.418,A -85,B 0,C 180,E1 -4784.745,E2 -4784.745} C_VEL
LIN {X 0,Y 525.125,Z 709.277,A -85,B 0,C 180,E1 -4786.124,E2 -4786.124} C_VEL
LIN {X 0,Y 525.668,Z 697.135,A -85,B 0,C 180,E1 -4787.407,E2 -4787.407} C_VEL
LIN {X 0,Y 526.337,Z 682.692,A -85,B 0,C 180,E1 -4788.692,E2 -4788.692} C_VEL
LIN {X 0,Y 526.999,Z 667.99,A -85,B 0,C 180,E1 -4789.78,E2 -4789.78} C_VEL
LIN {X 0,Y 527.615,Z 653.505,A -85,B 0,C 180,E1 -4790.671,E2 -4790.671} C_VEL
LIN {X 0,Y 528.229,Z 638.236,A -85,B 0,C 180,E1 -4791.441,E2 -4791.441} C_VEL
LIN {X 0,Y 528.782,Z 623.049,A -85,B 0,C 180,E1 -4792.052,E2 -4792.052} C_VEL
LIN {X 0,Y 529.114,Z 606.729,A -85,B 0,C 180,E1 -4792.547,E2 -4792.547} C_VEL
LIN {X 0,Y 529.189,Z 593.287,A -85,B 0,C 180,E1 -4792.844,E2 -4792.844} C_VEL
LIN {X 0,Y 524.794,Z 577.044,A -85,B 0,C 180,E1 -4793.324,E2 -4793.324} C_VEL
LIN {X 0,Y 525.265,Z 562.748,A -85,B 0,C 180,E1 -4796.63,E2 -4796.63} C_VEL
LIN {X 0,Y 525.665,Z 550.012,A -85,B 0,C 180,E1 -4799.654,E2 -4799.654} C_VEL
LIN {X 0,Y 526.13,Z 537.539,A -85,B 0,C 180,E1 -4802.697,E2 -4802.697} C_VEL
LIN {X 0,Y 526.422,Z 528.976,A -85,B 0,C 180,E1 -4804.802,E2 -4804.802} C_VEL
LIN {X 0,Y 526.395,Z 515.481,A -85,B 0,C 180,E1 -4807.649,E2 -4807.649} C_VEL
LIN {X 0,Y 526.195,Z 505.01,A -85,B 0,C 180,E1 -4809.874,E2 -4809.874} C_VEL
LIN {X 0,Y 523.97,Z 493.561,A -85,B 0,C 180,E1 -4812.569,E2 -4812.569} C_VEL
LIN {X 0,Y 523.943,Z 493.532,A -85,B 0,C 180,E1 -4815.773,E2 -4815.773} C_VEL
LIN {X 0,Y 523.943,Z 493.536,A -85,B 0,C 180,E1 -4818.908,E2 -4818.908} C_VEL
LIN {X 0,Y 523.918,Z 493.536,A -85,B 0,C 180,E1 -4821.899,E2 -4821.899} C_VEL
LIN {X 0,Y 523.937,Z 493.534,A -85,B 0,C 180,E1 -4824.91,E2 -4824.91} C_VEL
LIN {X 0,Y 523.939,Z 493.533,A -85,B 0,C 180,E1 -4827.68,E2 -4827.68} C_VEL
LIN {X 0,Y 523.956,Z 493.532,A -85,B 0,C 180,E1 -4830.677,E2 -4830.677} C_VEL
LIN {X 0,Y 523.977,Z 493.531,A -85,B 0,C 180,E1 -4833.729,E2 -4833.729} C_VEL
LIN {X 0,Y 523.941,Z 493.533,A -85,B 0,C 180,E1 -4836.899,E2 -4836.899} C_VEL
LIN {X 0,Y 523.939,Z 493.534,A -85,B 0,C 180,E1 -4836.952,E2 -4836.952} C_VEL
LIN {X 0,Y 525.813,Z 498.554,A -85,B 0,C 180,E1 -4837.15,E2 -4837.15} C_VEL
LIN {X 0,Y 529.163,Z 506.815,A -85,B 0,C 180,E1 -4837.5,E2 -4837.5} C_VEL
LIN {X 0,Y 528.709,Z 523.088,A -85,B 0,C 180,E1 -4837.994,E2 -4837.994} C_VEL
LIN {X 0,Y 528.182,Z 539.465,A -85,B 0,C 180,E1 -4838.658,E2 -4838.658} C_VEL
LIN {X 0,Y 527.582,Z 554.579,A -85,B 0,C 180,E1 -4839.431,E2 -4839.431} C_VEL
LIN {X 0,Y 526.974,Z 568.843,A -85,B 0,C 180,E1 -4840.322,E2 -4840.322} C_VEL
LIN {X 0,Y 526.344,Z 583.231,A -85,B 0,C 180,E1 -4841.401,E2 -4841.401} C_VEL
LIN {X 0,Y 525.734,Z 596.653,A -85,B 0,C 180,E1 -4842.596,E2 -4842.596} C_VEL
LIN {X 0,Y 525.126,Z 608.896,A -85,B 0,C 180,E1 -4843.877,E2 -4843.877} C_VEL
LIN {X 0,Y 524.71,Z 620.132,A -85,B 0,C 180,E1 -4845.257,E2 -4845.257} C_VEL
LIN {X 0,Y 524.235,Z 629.721,A -85,B 0,C 180,E1 -4846.629,E2 -4846.629} C_VEL
LIN {X 0,Y 523.959,Z 639.468,A -85,B 0,C 180,E1 -4848.285,E2 -4848.285} C_VEL
LIN {X 0,Y 523.661,Z 647.636,A -85,B 0,C 180,E1 -4849.952,E2 -4849.952} C_VEL
LIN {X 0,Y 523.528,Z 653.899,A -85,B 0,C 180,E1 -4851.509,E2 -4851.509} C_VEL
LIN {X 0,Y 523.48,Z 658.995,A -85,B 0,C 180,E1 -4853.06,E2 -4853.06} C_VEL
LIN {X 0,Y 523.399,Z 662.971,A -85,B 0,C 180,E1 -4854.607,E2 -4854.607} C_VEL
LIN {X 0,Y 523.399,Z 665.917,A -85,B 0,C 180,E1 -4856.151,E2 -4856.151} C_VEL
LIN {X 0,Y 523.327,Z 667.875,A -85,B 0,C 180,E1 -4857.691,E2 -4857.691} C_VEL
LIN {X 0,Y 523.248,Z 668.858,A -85,B 0,C 180,E1 -4859.231,E2 -4859.231} C_VEL
LIN {X 0,Y 523.247,Z 668.875,A -85,B 0,C 180,E1 -4860.77,E2 -4860.77} C_VEL
LIN {X 0,Y 523.327,Z 667.949,A -85,B 0,C 180,E1 -4862.309,E2 -4862.309} C_VEL
LIN {X 0,Y 523.401,Z 666.054,A -85,B 0,C 180,E1 -4863.85,E2 -4863.85} C_VEL
LIN {X 0,Y 523.399,Z 663.167,A -85,B 0,C 180,E1 -4865.394,E2 -4865.394} C_VEL
LIN {X 0,Y 523.481,Z 659.267,A -85,B 0,C 180,E1 -4866.94,E2 -4866.94} C_VEL
LIN {X 0,Y 523.526,Z 654.24,A -85,B 0,C 180,E1 -4868.492,E2 -4868.492} C_VEL
LIN {X 0,Y 523.656,Z 648.053,A -85,B 0,C 180,E1 -4870.048,E2 -4870.048} C_VEL
LIN {X 0,Y 523.919,Z 640.077,A -85,B 0,C 180,E1 -4871.694,E2 -4871.694} C_VEL
LIN {X 0,Y 524.245,Z 630.261,A -85,B 0,C 180,E1 -4873.371,E2 -4873.371} C_VEL
LIN {X 0,Y 524.719,Z 619.726,A -85,B 0,C 180,E1 -4874.885,E2 -4874.885} C_VEL
LIN {X 0,Y 525.172,Z 607.951,A -85,B 0,C 180,E1 -4876.322,E2 -4876.322} C_VEL
LIN {X 0,Y 525.704,Z 595.534,A -85,B 0,C 180,E1 -4877.606,E2 -4877.606} C_VEL
LIN {X 0,Y 526.382,Z 581.99,A -85,B 0,C 180,E1 -4878.791,E2 -4878.791} C_VEL
LIN {X 0,Y 527.073,Z 567.17,A -85,B 0,C 180,E1 -4879.878,E2 -4879.878} C_VEL
LIN {X 0,Y 527.613,Z 554.311,A -85,B 0,C 180,E1 -4880.671,E2 -4880.671} C_VEL
LIN {X 0,Y 528.223,Z 539.006,A -85,B 0,C 180,E1 -4881.451,E2 -4881.451} C_VEL
LIN {X 0,Y 528.756,Z 520.98,A -85,B 0,C 180,E1 -4882.166,E2 -4882.166} C_VEL
LIN {X 0,Y 529.072,Z 506.245,A -85,B 0,C 180,E1 -4882.6,E2 -4882.6} C_VEL
LIN {X 0,Y 523.986,Z 493.941,A -85,B 0,C 180,E1 -4883.111,E2 -4883.111} C_VEL
LIN {X 0,Y 523.936,Z 493.538,A -85,B 0,C 180,E1 -4883.128,E2 -4883.128} C_VEL
LIN {X 0,Y 523.977,Z 493.53,A -85,B 0,C 180,E1 -4886.272,E2 -4886.272} C_VEL
LIN {X 0,Y 523.958,Z 493.532,A -85,B 0,C 180,E1 -4889.324,E2 -4889.324} C_VEL
LIN {X 0,Y 523.939,Z 493.534,A -85,B 0,C 180,E1 -4892.32,E2 -4892.32} C_VEL
LIN {X 0,Y 523.938,Z 493.533,A -85,B 0,C 180,E1 -4895.226,E2 -4895.226} C_VEL
LIN {X 0,Y 523.913,Z 493.537,A -85,B 0,C 180,E1 -4897.866,E2 -4897.866} C_VEL
LIN {X 0,Y 523.255,Z 493.62,A -85,B 0,C 180,E1 -4898.508,E2 -4898.508} C_VEL
LIN {X 0,Y 520.393,Z 493.975,A -85,B 0,C 180,E1 -4899.549,E2 -4899.549} C_VEL
LIN {X 0,Y 517.98,Z 494.28,A -85,B 0,C 180,E1 -4900.388,E2 -4900.388} C_VEL
LIN {X 0,Y 516.964,Z 494.403,A -85,B 0,C 180,E1 -4901.036,E2 -4901.036} C_VEL
LIN {X 0,Y 516.891,Z 494.411,A -85,B 0,C 180,E1 -4901.256,E2 -4901.256} C_VEL
LIN {X 0,Y 516.887,Z 494.411,A -85,B 0,C 180,E1 -4903.903,E2 -4903.903} C_VEL
LIN {X 0,Y 516.888,Z 494.415,A -85,B 0,C 180,E1 -4906.107,E2 -4906.107} C_VEL
LIN {X 0,Y 516.923,Z 494.407,A -85,B 0,C 180,E1 -4908.398,E2 -4908.398} C_VEL
LIN {X 0,Y 516.887,Z 494.412,A -85,B 0,C 180,E1 -4911.284,E2 -4911.284} C_VEL
LIN {X 0,Y 516.876,Z 494.415,A -85,B 0,C 180,E1 -4914.22,E2 -4914.22} C_VEL
LIN {X 0,Y 516.901,Z 494.413,A -85,B 0,C 180,E1 -4917.053,E2 -4917.053} C_VEL
LIN {X 0,Y 516.898,Z 494.413,A -85,B 0,C 180,E1 -4919.796,E2 -4919.796} C_VEL
LIN {X 0,Y 516.932,Z 494.407,A -85,B 0,C 180,E1 -4922.467,E2 -4922.467} C_VEL
LIN {X 0,Y 517.012,Z 494.421,A -85,B 0,C 180,E1 -4925.612,E2 -4925.612} C_VEL
LIN {X 0,Y 516.923,Z 499.724,A -85,B 0,C 180,E1 -4928.463,E2 -4928.463} C_VEL
LIN {X 0,Y 516.882,Z 504.184,A -85,B 0,C 180,E1 -4930.953,E2 -4930.953} C_VEL
LIN {X 0,Y 516.836,Z 508.48,A -85,B 0,C 180,E1 -4933.407,E2 -4933.407} C_VEL
LIN {X 0,Y 516.773,Z 512.634,A -85,B 0,C 180,E1 -4935.83,E2 -4935.83} C_VEL
LIN {X 0,Y 516.725,Z 518.033,A -85,B 0,C 180,E1 -4939.022,E2 -4939.022} C_VEL
LIN {X 0,Y 516.607,Z 521.918,A -85,B 0,C 180,E1 -4941.416,E2 -4941.416} C_VEL
LIN {X 0,Y 522.691,Z 541.846,A -85,B 0,C 180,E1 -4942.085,E2 -4942.085} C_VEL
LIN {X 0,Y 522.321,Z 556.477,A -85,B 0,C 180,E1 -4942.486,E2 -4942.486} C_VEL
LIN {X 0,Y 521.852,Z 569.973,A -85,B 0,C 180,E1 -4942.968,E2 -4942.968} C_VEL
LIN {X 0,Y 521.338,Z 582.419,A -85,B 0,C 180,E1 -4943.517,E2 -4943.517} C_VEL
LIN {X 0,Y 520.839,Z 595.073,A -85,B 0,C 180,E1 -4944.191,E2 -4944.191} C_VEL
LIN {X 0,Y 520.292,Z 607.36,A -85,B 0,C 180,E1 -4944.962,E2 -4944.962} C_VEL
LIN {X 0,Y 519.705,Z 619.243,A -85,B 0,C 180,E1 -4945.831,E2 -4945.831} C_VEL
LIN {X 0,Y 519.029,Z 632.87,A -85,B 0,C 180,E1 -4946.992,E2 -4946.992} C_VEL
LIN {X 0,Y 518.402,Z 645.25,A -85,B 0,C 180,E1 -4948.251,E2 -4948.251} C_VEL
LIN {X 0,Y 517.891,Z 655.179,A -85,B 0,C 180,E1 -4949.416,E2 -4949.416} C_VEL
LIN {X 0,Y 517.418,Z 663.899,A -85,B 0,C 180,E1 -4950.583,E2 -4950.583} C_VEL
LIN {X 0,Y 517.123,Z 672.752,A -85,B 0,C 180,E1 -4951.946,E2 -4951.946} C_VEL
LIN {X 0,Y 516.801,Z 680.42,A -85,B 0,C 180,E1 -4953.312,E2 -4953.312} C_VEL
LIN {X 0,Y 516.638,Z 687.002,A -85,B 0,C 180,E1 -4954.681,E2 -4954.681} C_VEL
LIN {X 0,Y 516.472,Z 693.393,A -85,B 0,C 180,E1 -4956.249,E2 -4956.249} C_VEL
LIN {X 0,Y 516.37,Z 699.683,A -85,B 0,C 180,E1 -4958.215,E2 -4958.215} C_VEL
LIN {X 0,Y 516.22,Z 702.695,A -85,B 0,C 180,E1 -4959.402,E2 -4959.402} C_VEL
LIN {X 0,Y 516.257,Z 705.726,A -85,B 0,C 180,E1 -4960.986,E2 -4960.986} C_VEL
LIN {X 0,Y 516.175,Z 707.762,A -85,B 0,C 180,E1 -4962.582,E2 -4962.582} C_VEL
LIN {X 0,Y 516.173,Z 708.79,A -85,B 0,C 180,E1 -4964.186,E2 -4964.186} C_VEL
LIN {X 0,Y 516.131,Z 708.819,A -85,B 0,C 180,E1 -4965.802,E2 -4965.802} C_VEL
LIN {X 0,Y 516.202,Z 707.831,A -85,B 0,C 180,E1 -4967.428,E2 -4967.428} C_VEL
LIN {X 0,Y 516.172,Z 705.772,A -85,B 0,C 180,E1 -4969.072,E2 -4969.072} C_VEL
LIN {X 0,Y 516.254,Z 702.605,A -85,B 0,C 180,E1 -4970.728,E2 -4970.728} C_VEL
LIN {X 0,Y 516.351,Z 698.185,A -85,B 0,C 180,E1 -4972.401,E2 -4972.401} C_VEL
LIN {X 0,Y 516.485,Z 692.423,A -85,B 0,C 180,E1 -4974.092,E2 -4974.092} C_VEL
LIN {X 0,Y 516.604,Z 687.168,A -85,B 0,C 180,E1 -4975.373,E2 -4975.373} C_VEL
LIN {X 0,Y 516.847,Z 679.883,A -85,B 0,C 180,E1 -4976.879,E2 -4976.879} C_VEL
LIN {X 0,Y 517.085,Z 672.866,A -85,B 0,C 180,E1 -4978.126,E2 -4978.126} C_VEL
LIN {X 0,Y 517.495,Z 664.232,A -85,B 0,C 180,E1 -4979.456,E2 -4979.456} C_VEL
LIN {X 0,Y 517.956,Z 654.113,A -85,B 0,C 180,E1 -4980.81,E2 -4980.81} C_VEL
LIN {X 0,Y 518.602,Z 641.447,A -85,B 0,C 180,E1 -4982.248,E2 -4982.248} C_VEL
LIN {X 0,Y 519.144,Z 630.278,A -85,B 0,C 180,E1 -4983.329,E2 -4983.329} C_VEL
LIN {X 0,Y 519.745,Z 618.294,A -85,B 0,C 180,E1 -4984.332,E2 -4984.332} C_VEL
LIN {X 0,Y 520.299,Z 607.013,A -85,B 0,C 180,E1 -4985.152,E2 -4985.152} C_VEL
LIN {X 0,Y 520.809,Z 596.093,A -85,B 0,C 180,E1 -4985.84,E2 -4985.84} C_VEL
LIN {X 0,Y 521.295,Z 583.846,A -85,B 0,C 180,E1 -4986.503,E2 -4986.503} C_VEL
LIN {X 0,Y 521.779,Z 571.391,A -85,B 0,C 180,E1 -4987.066,E2 -4987.066} C_VEL
LIN {X 0,Y 522.223,Z 558.957,A -85,B 0,C 180,E1 -4987.524,E2 -4987.524} C_VEL
LIN {X 0,Y 522.583,Z 546.843,A -85,B 0,C 180,E1 -4987.879,E2 -4987.879} C_VEL
LIN {X 0,Y 522.591,Z 541.703,A -85,B 0,C 180,E1 -4988.014,E2 -4988.014} C_VEL
LIN {X 0,Y 516.53,Z 521.947,A -85,B 0,C 180,E1 -4988.678,E2 -4988.678} C_VEL
LIN {X 0,Y 516.678,Z 517.007,A -85,B 0,C 180,E1 -4991.797,E2 -4991.797} C_VEL
LIN {X 0,Y 516.784,Z 511.467,A -85,B 0,C 180,E1 -4995.003,E2 -4995.003} C_VEL
LIN {X 0,Y 516.837,Z 507.485,A -85,B 0,C 180,E1 -4997.246,E2 -4997.246} C_VEL
LIN {X 0,Y 516.908,Z 502.126,A -85,B 0,C 180,E1 -5000.281,E2 -5000.281} C_VEL
LIN {X 0,Y 516.953,Z 496.45,A -85,B 0,C 180,E1 -5003.329,E2 -5003.329} C_VEL
LIN {X 0,Y 516.954,Z 494.407,A -85,B 0,C 180,E1 -5004.476,E2 -5004.476} C_VEL
LIN {X 0,Y 516.894,Z 494.414,A -85,B 0,C 180,E1 -5007.454,E2 -5007.454} C_VEL
LIN {X 0,Y 516.928,Z 494.41,A -85,B 0,C 180,E1 -5010.695,E2 -5010.695} C_VEL
LIN {X 0,Y 516.937,Z 494.408,A -85,B 0,C 180,E1 -5013.802,E2 -5013.802} C_VEL
LIN {X 0,Y 516.884,Z 494.412,A -85,B 0,C 180,E1 -5016.777,E2 -5016.777} C_VEL
LIN {X 0,Y 516.93,Z 494.408,A -85,B 0,C 180,E1 -5019.73,E2 -5019.73} C_VEL
LIN {X 0,Y 516.922,Z 494.409,A -85,B 0,C 180,E1 -5022.596,E2 -5022.596} C_VEL
LIN {X 0,Y 516.931,Z 494.407,A -85,B 0,C 180,E1 -5025.029,E2 -5025.029} C_VEL
LIN {X 0,Y 516.994,Z 494.401,A -85,B 0,C 180,E1 -5028.234,E2 -5028.234} C_VEL
LIN {X 0,Y 516.963,Z 494.402,A -85,B 0,C 180,E1 -5031.399,E2 -5031.399} C_VEL
LIN {X 0,Y 517.056,Z 494.39,A -85,B 0,C 180,E1 -5034.54,E2 -5034.54} C_VEL
LIN {X 0,Y 517.078,Z 494.389,A -85,B 0,C 180,E1 -5037.663,E2 -5037.663} C_VEL
LIN {X 0,Y 517.086,Z 494.389,A -85,B 0,C 180,E1 -5040.778,E2 -5040.778} C_VEL
LIN {X 0,Y 517.008,Z 494.397,A -85,B 0,C 180,E1 -5043.117,E2 -5043.117} C_VEL
LIN {X 0,Y 517,Z 494.4,A -85,B 0,C 180,E1 -5046.243,E2 -5046.243} C_VEL
LIN {X 0,Y 516.948,Z 494.402,A -85,B 0,C 180,E1 -5049.389,E2 -5049.389} C_VEL
LIN {X 0,Y 516.971,Z 494.399,A -85,B 0,C 180,E1 -5051.824,E2 -5051.824} C_VEL
LIN {X 0,Y 516.932,Z 494.405,A -85,B 0,C 180,E1 -5055.147,E2 -5055.147} C_VEL
LIN {X 0,Y 516.914,Z 494.395,A -85,B 0,C 180,E1 -5058.222,E2 -5058.222} C_VEL
LIN {X 0,Y 516.904,Z 494.41,A -85,B 0,C 180,E1 -5060.701,E2 -5060.701} C_VEL
LIN {X 0,Y 516.881,Z 494.408,A -85,B 0,C 180,E1 -5063.223,E2 -5063.223} C_VEL
LIN {X 0,Y 516.934,Z 494.402,A -85,B 0,C 180,E1 -5066.197,E2 -5066.197} C_VEL
LIN {X 0,Y 516.925,Z 494.41,A -85,B 0,C 180,E1 -5069.304,E2 -5069.304} C_VEL
LIN {X 0,Y 516.891,Z 494.411,A -85,B 0,C 180,E1 -5072.545,E2 -5072.545} C_VEL
LIN {X 0,Y 516.874,Z 494.412,A -85,B 0,C 180,E1 -5075.333,E2 -5075.333} C_VEL
LIN {X 0,Y 516.876,Z 494.413,A -85,B 0,C 180,E1 -5077.945,E2 -5077.945} C_VEL
LIN {X 0,Y 516.907,Z 494.408,A -85,B 0,C 180,E1 -5080.739,E2 -5080.739} C_VEL
LIN {X 0,Y 516.873,Z 494.416,A -85,B 0,C 180,E1 -5083.904,E2 -5083.904} C_VEL
LIN {X 0,Y 516.902,Z 494.483,A -85,B 0,C 180,E1 -5085.614,E2 -5085.614} C_VEL
LIN {X 0,Y 519.05,Z 504.238,A -85,B 0,C 180,E1 -5088.437,E2 -5088.437} C_VEL
LIN {X 0,Y 519.905,Z 508.221,A -85,B 0,C 180,E1 -5089.546,E2 -5089.546} C_VEL
LIN {X 0,Y 519.973,Z 516.044,A -85,B 0,C 180,E1 -5091.558,E2 -5091.558} C_VEL
LIN {X 0,Y 519.652,Z 527.677,A -85,B 0,C 180,E1 -5094.442,E2 -5094.442} C_VEL
LIN {X 0,Y 519.268,Z 539.142,A -85,B 0,C 180,E1 -5097.224,E2 -5097.224} C_VEL
LIN {X 0,Y 518.711,Z 552.252,A -85,B 0,C 180,E1 -5100.459,E2 -5100.459} C_VEL
LIN {X 0,Y 518.298,Z 564.57,A -85,B 0,C 180,E1 -5103.42,E2 -5103.42} C_VEL
LIN {X 0,Y 517.89,Z 577.221,A -85,B 0,C 180,E1 -5106.372,E2 -5106.372} C_VEL
LIN {X 0,Y 522.752,Z 594.996,A -85,B 0,C 180,E1 -5106.888,E2 -5106.888} C_VEL
LIN {X 0,Y 522.478,Z 611.542,A -85,B 0,C 180,E1 -5107.288,E2 -5107.288} C_VEL
LIN {X 0,Y 521.972,Z 628.27,A -85,B 0,C 180,E1 -5107.853,E2 -5107.853} C_VEL
LIN {X 0,Y 521.348,Z 643.289,A -85,B 0,C 180,E1 -5108.51,E2 -5108.51} C_VEL
LIN {X 0,Y 520.706,Z 658.733,A -85,B 0,C 180,E1 -5109.354,E2 -5109.354} C_VEL
LIN {X 0,Y 520.025,Z 673.695,A -85,B 0,C 180,E1 -5110.357,E2 -5110.357} C_VEL
LIN {X 0,Y 519.302,Z 687.606,A -85,B 0,C 180,E1 -5111.475,E2 -5111.475} C_VEL
LIN {X 0,Y 518.653,Z 700.079,A -85,B 0,C 180,E1 -5112.657,E2 -5112.657} C_VEL
LIN {X 0,Y 518.058,Z 712.643,A -85,B 0,C 180,E1 -5114.056,E2 -5114.056} C_VEL
LIN {X 0,Y 517.556,Z 723.344,A -85,B 0,C 180,E1 -5115.452,E2 -5115.452} C_VEL
LIN {X 0,Y 517.1,Z 733.678,A -85,B 0,C 180,E1 -5117.042,E2 -5117.042} C_VEL
LIN {X 0,Y 516.819,Z 742.289,A -85,B 0,C 180,E1 -5118.629,E2 -5118.629} C_VEL
LIN {X 0,Y 516.55,Z 749.494,A -85,B 0,C 180,E1 -5120.209,E2 -5120.209} C_VEL
LIN {X 0,Y 516.418,Z 755.469,A -85,B 0,C 180,E1 -5121.785,E2 -5121.785} C_VEL
LIN {X 0,Y 516.32,Z 761.25,A -85,B 0,C 180,E1 -5123.749,E2 -5123.749} C_VEL
LIN {X 0,Y 516.225,Z 764.638,A -85,B 0,C 180,E1 -5125.315,E2 -5125.315} C_VEL
LIN {X 0,Y 516.267,Z 767.091,A -85,B 0,C 180,E1 -5126.879,E2 -5126.879} C_VEL
LIN {X 0,Y 516.188,Z 768.48,A -85,B 0,C 180,E1 -5128.44,E2 -5128.44} C_VEL
LIN {X 0,Y 516.149,Z 769,A -85,B 0,C 180,E1 -5130.001,E2 -5130.001} C_VEL
LIN {X 0,Y 516.188,Z 768.479,A -85,B 0,C 180,E1 -5131.561,E2 -5131.561} C_VEL
LIN {X 0,Y 516.267,Z 767.088,A -85,B 0,C 180,E1 -5133.122,E2 -5133.122} C_VEL
LIN {X 0,Y 516.226,Z 764.634,A -85,B 0,C 180,E1 -5134.686,E2 -5134.686} C_VEL
LIN {X 0,Y 516.369,Z 760.555,A -85,B 0,C 180,E1 -5136.508,E2 -5136.508} C_VEL
LIN {X 0,Y 516.419,Z 755.465,A -85,B 0,C 180,E1 -5138.216,E2 -5138.216} C_VEL
LIN {X 0,Y 516.62,Z 747.853,A -85,B 0,C 180,E1 -5140.187,E2 -5140.187} C_VEL
LIN {X 0,Y 516.915,Z 740.159,A -85,B 0,C 180,E1 -5141.788,E2 -5141.788} C_VEL
LIN {X 0,Y 517.205,Z 731.207,A -85,B 0,C 180,E1 -5143.357,E2 -5143.357} C_VEL
LIN {X 0,Y 517.735,Z 720.417,A -85,B 0,C 180,E1 -5144.947,E2 -5144.947} C_VEL
LIN {X 0,Y 518.143,Z 711,A -85,B 0,C 180,E1 -5146.145,E2 -5146.145} C_VEL
LIN {X 0,Y 518.643,Z 700.062,A -85,B 0,C 180,E1 -5147.345,E2 -5147.345} C_VEL
LIN {X 0,Y 519.31,Z 686.537,A -85,B 0,C 180,E1 -5148.618,E2 -5148.618} C_VEL
LIN {X 0,Y 520.073,Z 672.259,A -85,B 0,C 180,E1 -5149.746,E2 -5149.746} C_VEL
LIN {X 0,Y 520.767,Z 657.015,A -85,B 0,C 180,E1 -5150.748,E2 -5150.748} C_VEL
LIN {X 0,Y 521.476,Z 640.833,A -85,B 0,C 180,E1 -5151.612,E2 -5151.612} C_VEL
LIN {X 0,Y 522.045,Z 626.317,A -85,B 0,C 180,E1 -5152.222,E2 -5152.222} C_VEL
LIN {X 0,Y 522.506,Z 610.625,A -85,B 0,C 180,E1 -5152.737,E2 -5152.737} C_VEL
LIN {X 0,Y 522.612,Z 594.639,A -85,B 0,C 180,E1 -5153.125,E2 -5153.125} C_VEL
LIN {X 0,Y 517.846,Z 577.05,A -85,B 0,C 180,E1 -5153.654,E2 -5153.654} C_VEL
LIN {X 0,Y 518.304,Z 564.562,A -85,B 0,C 180,E1 -5156.582,E2 -5156.582} C_VEL
LIN {X 0,Y 518.719,Z 552.245,A -85,B 0,C 180,E1 -5159.542,E2 -5159.542} C_VEL
LIN {X 0,Y 519.276,Z 539.135,A -85,B 0,C 180,E1 -5162.777,E2 -5162.777} C_VEL
LIN {X 0,Y 519.331,Z 533.753,A -85,B 0,C 180,E1 -5164.031,E2 -5164.031} C_VEL
LIN {X 0,Y 519.431,Z 520.796,A -85,B 0,C 180,E1 -5166.78,E2 -5166.78} C_VEL
LIN {X 0,Y 519.329,Z 508.045,A -85,B 0,C 180,E1 -5169.523,E2 -5169.523} C_VEL
LIN {X 0,Y 518.422,Z 502.063,A -85,B 0,C 180,E1 -5170.907,E2 -5170.907} C_VEL
LIN {X 0,Y 516.917,Z 494.412,A -85,B 0,C 180,E1 -5172.828,E2 -5172.828} C_VEL
LIN {X 0,Y 516.924,Z 494.41,A -85,B 0,C 180,E1 -5175.011,E2 -5175.011} C_VEL
LIN {X 0,Y 516.916,Z 494.411,A -85,B 0,C 180,E1 -5178.399,E2 -5178.399} C_VEL
LIN {X 0,Y 516.884,Z 494.412,A -85,B 0,C 180,E1 -5181.285,E2 -5181.285} C_VEL
LIN {X 0,Y 516.889,Z 494.414,A -85,B 0,C 180,E1 -5184.221,E2 -5184.221} C_VEL
LIN {X 0,Y 516.897,Z 494.41,A -85,B 0,C 180,E1 -5187.054,E2 -5187.054} C_VEL
LIN {X 0,Y 516.893,Z 494.413,A -85,B 0,C 180,E1 -5189.797,E2 -5189.797} C_VEL
LIN {X 0,Y 516.93,Z 494.408,A -85,B 0,C 180,E1 -5192.468,E2 -5192.468} C_VEL
LIN {X 0,Y 516.912,Z 494.408,A -85,B 0,C 180,E1 -5195.072,E2 -5195.072} C_VEL
LIN {X 0,Y 516.898,Z 494.412,A -85,B 0,C 180,E1 -5196.659,E2 -5196.659} C_VEL
LIN {X 0,Y 518.849,Z 499.57,A -85,B 0,C 180,E1 -5196.86,E2 -5196.86} C_VEL
LIN {X 0,Y 522.561,Z 508.456,A -85,B 0,C 180,E1 -5197.245,E2 -5197.245} C_VEL
LIN {X 0,Y 522.076,Z 525.01,A -85,B 0,C 180,E1 -5197.772,E2 -5197.772} C_VEL
LIN {X 0,Y 521.497,Z 541.089,A -85,B 0,C 180,E1 -5198.447,E2 -5198.447} C_VEL
LIN {X 0,Y 520.831,Z 556.288,A -85,B 0,C 180,E1 -5199.255,E2 -5199.255} C_VEL
LIN {X 0,Y 520.1,Z 571.659,A -85,B 0,C 180,E1 -5200.256,E2 -5200.256} C_VEL
LIN {X 0,Y 519.348,Z 586.008,A -85,B 0,C 180,E1 -5201.378,E2 -5201.378} C_VEL
LIN {X 0,Y 518.693,Z 599.685,A -85,B 0,C 180,E1 -5202.658,E2 -5202.658} C_VEL
LIN {X 0,Y 518.06,Z 612.284,A -85,B 0,C 180,E1 -5204.056,E2 -5204.056} C_VEL
LIN {X 0,Y 517.565,Z 623.009,A -85,B 0,C 180,E1 -5205.451,E2 -5205.451} C_VEL
LIN {X 0,Y 517.111,Z 633.396,A -85,B 0,C 180,E1 -5207.042,E2 -5207.042} C_VEL
LIN {X 0,Y 516.824,Z 642.095,A -85,B 0,C 180,E1 -5208.628,E2 -5208.628} C_VEL
LIN {X 0,Y 516.556,Z 649.337,A -85,B 0,C 180,E1 -5210.209,E2 -5210.209} C_VEL
LIN {X 0,Y 516.421,Z 655.314,A -85,B 0,C 180,E1 -5211.785,E2 -5211.785} C_VEL
LIN {X 0,Y 516.371,Z 660.469,A -85,B 0,C 180,E1 -5213.493,E2 -5213.493} C_VEL
LIN {X 0,Y 516.227,Z 664.563,A -85,B 0,C 180,E1 -5215.315,E2 -5215.315} C_VEL
LIN {X 0,Y 516.271,Z 667.019,A -85,B 0,C 180,E1 -5216.879,E2 -5216.879} C_VEL
LIN {X 0,Y 516.186,Z 668.481,A -85,B 0,C 180,E1 -5218.44,E2 -5218.44} C_VEL
LIN {X 0,Y 516.152,Z 668.997,A -85,B 0,C 180,E1 -5220,E2 -5220} C_VEL
LIN {X 0,Y 516.186,Z 668.532,A -85,B 0,C 180,E1 -5221.561,E2 -5221.561} C_VEL
LIN {X 0,Y 516.272,Z 667.122,A -85,B 0,C 180,E1 -5223.122,E2 -5223.122} C_VEL
LIN {X 0,Y 516.227,Z 664.733,A -85,B 0,C 180,E1 -5224.686,E2 -5224.686} C_VEL
LIN {X 0,Y 516.372,Z 660.684,A -85,B 0,C 180,E1 -5226.507,E2 -5226.507} C_VEL
LIN {X 0,Y 516.421,Z 655.591,A -85,B 0,C 180,E1 -5228.216,E2 -5228.216} C_VEL
LIN {X 0,Y 516.549,Z 649.68,A -85,B 0,C 180,E1 -5229.792,E2 -5229.792} C_VEL
LIN {X 0,Y 516.786,Z 642.517,A -85,B 0,C 180,E1 -5231.373,E2 -5231.373} C_VEL
LIN {X 0,Y 517.095,Z 633.91,A -85,B 0,C 180,E1 -5232.96,E2 -5232.96} C_VEL
LIN {X 0,Y 517.55,Z 623.652,A -85,B 0,C 180,E1 -5234.55,E2 -5234.55} C_VEL
LIN {X 0,Y 518.027,Z 613.044,A -85,B 0,C 180,E1 -5235.946,E2 -5235.946} C_VEL
LIN {X 0,Y 518.642,Z 600.53,A -85,B 0,C 180,E1 -5237.345,E2 -5237.345} C_VEL
LIN {X 0,Y 519.262,Z 588.102,A -85,B 0,C 180,E1 -5238.527,E2 -5238.527} C_VEL
LIN {X 0,Y 519.97,Z 574.233,A -85,B 0,C 180,E1 -5239.647,E2 -5239.647} C_VEL
LIN {X 0,Y 520.658,Z 559.388,A -85,B 0,C 180,E1 -5240.649,E2 -5240.649} C_VEL
LIN {X 0,Y 521.337,Z 544.433,A -85,B 0,C 180,E1 -5241.479,E2 -5241.479} C_VEL
LIN {X 0,Y 521.866,Z 530.45,A -85,B 0,C 180,E1 -5242.102,E2 -5242.102} C_VEL
LIN {X 0,Y 522.31,Z 516.967,A -85,B 0,C 180,E1 -5242.588,E2 -5242.588} C_VEL
LIN {X 0,Y 522.428,Z 508.112,A -85,B 0,C 180,E1 -5242.854,E2 -5242.854} C_VEL
LIN {X 0,Y 517.011,Z 495.168,A -85,B 0,C 180,E1 -5243.408,E2 -5243.408} C_VEL
LIN {X 0,Y 516.883,Z 494.416,A -85,B 0,C 180,E1 -5243.44,E2 -5243.44} C_VEL
LIN {X 0,Y 516.946,Z 494.406,A -85,B 0,C 180,E1 -5246.196,E2 -5246.196} C_VEL
LIN {X 0,Y 516.926,Z 494.408,A -85,B 0,C 180,E1 -5249.305,E2 -5249.305} C_VEL
LIN {X 0,Y 516.9,Z 494.41,A -85,B 0,C 180,E1 -5252.543,E2 -5252.543} C_VEL
LIN {X 0,Y 516.885,Z 494.412,A -85,B 0,C 180,E1 -5255.332,E2 -5255.332} C_VEL
LIN {X 0,Y 516.886,Z 494.412,A -85,B 0,C 180,E1 -5257.943,E2 -5257.943} C_VEL
LIN {X 0,Y 516.887,Z 494.412,A -85,B 0,C 180,E1 -5260.742,E2 -5260.742} C_VEL
LIN {X 0,Y 516.891,Z 494.411,A -85,B 0,C 180,E1 -5261.256,E2 -5261.256} C_VEL
LIN {X 0,Y 516.255,Z 494.495,A -85,B 0,C 180,E1 -5261.906,E2 -5261.906} C_VEL
LIN {X 0,Y 513.415,Z 494.854,A -85,B 0,C 180,E1 -5262.962,E2 -5262.962} C_VEL
LIN {X 0,Y 510.988,Z 495.156,A -85,B 0,C 180,E1 -5263.813,E2 -5263.813} C_VEL
LIN {X 0,Y 509.934,Z 495.283,A -85,B 0,C 180,E1 -5264.47,E2 -5264.47} C_VEL
LIN {X 0,Y 509.843,Z 495.292,A -85,B 0,C 180,E1 -5264.692,E2 -5264.692} C_VEL
LIN {X 0,Y 509.864,Z 495.286,A -85,B 0,C 180,E1 -5268.103,E2 -5268.103} C_VEL
LIN {X 0,Y 509.852,Z 495.29,A -85,B 0,C 180,E1 -5270.648,E2 -5270.648} C_VEL
LIN {X 0,Y 509.83,Z 495.293,A -85,B 0,C 180,E1 -5273.647,E2 -5273.647} C_VEL
LIN {X 0,Y 509.865,Z 495.289,A -85,B 0,C 180,E1 -5276.539,E2 -5276.539} C_VEL
LIN {X 0,Y 509.851,Z 495.291,A -85,B 0,C 180,E1 -5279.334,E2 -5279.334} C_VEL
LIN {X 0,Y 509.896,Z 495.285,A -85,B 0,C 180,E1 -5282.054,E2 -5282.054} C_VEL
LIN {X 0,Y 509.91,Z 495.286,A -85,B 0,C 180,E1 -5284.705,E2 -5284.705} C_VEL
LIN {X 0,Y 509.984,Z 495.388,A -85,B 0,C 180,E1 -5285.579,E2 -5285.579} C_VEL
LIN {X 0,Y 509.881,Z 500.174,A -85,B 0,C 180,E1 -5288.151,E2 -5288.151} C_VEL
LIN {X 0,Y 509.879,Z 504.705,A -85,B 0,C 180,E1 -5290.682,E2 -5290.682} C_VEL
LIN {X 0,Y 509.82,Z 509.058,A -85,B 0,C 180,E1 -5293.172,E2 -5293.172} C_VEL
LIN {X 0,Y 509.755,Z 513.276,A -85,B 0,C 180,E1 -5295.63,E2 -5295.63} C_VEL
LIN {X 0,Y 509.706,Z 518.693,A -85,B 0,C 180,E1 -5298.869,E2 -5298.869} C_VEL
LIN {X 0,Y 509.57,Z 522.488,A -85,B 0,C 180,E1 -5301.08,E2 -5301.08} C_VEL
LIN {X 0,Y 515.24,Z 540.362,A -85,B 0,C 180,E1 -5301.688,E2 -5301.688} C_VEL
LIN {X 0,Y 516.158,Z 544.294,A -85,B 0,C 180,E1 -5301.834,E2 -5301.834} C_VEL
LIN {X 0,Y 515.688,Z 558.976,A -85,B 0,C 180,E1 -5302.259,E2 -5302.259} C_VEL
LIN {X 0,Y 515.186,Z 572.289,A -85,B 0,C 180,E1 -5302.761,E2 -5302.761} C_VEL
LIN {X 0,Y 514.577,Z 586.533,A -85,B 0,C 180,E1 -5303.431,E2 -5303.431} C_VEL
LIN {X 0,Y 513.809,Z 603.189,A -85,B 0,C 180,E1 -5304.406,E2 -5304.406} C_VEL
LIN {X 0,Y 513.155,Z 615.614,A -85,B 0,C 180,E1 -5305.286,E2 -5305.286} C_VEL
LIN {X 0,Y 512.574,Z 626.406,A -85,B 0,C 180,E1 -5306.167,E2 -5306.167} C_VEL
LIN {X 0,Y 512.035,Z 635.952,A -85,B 0,C 180,E1 -5307.049,E2 -5307.049} C_VEL
LIN {X 0,Y 511.417,Z 647.066,A -85,B 0,C 180,E1 -5308.227,E2 -5308.227} C_VEL
LIN {X 0,Y 510.957,Z 655.268,A -85,B 0,C 180,E1 -5309.211,E2 -5309.211} C_VEL
LIN {X 0,Y 510.453,Z 663.979,A -85,B 0,C 180,E1 -5310.394,E2 -5310.394} C_VEL
LIN {X 0,Y 510.119,Z 671.653,A -85,B 0,C 180,E1 -5311.578,E2 -5311.578} C_VEL
LIN {X 0,Y 509.792,Z 679.452,A -85,B 0,C 180,E1 -5312.962,E2 -5312.962} C_VEL
LIN {X 0,Y 509.598,Z 686.164,A -85,B 0,C 180,E1 -5314.349,E2 -5314.349} C_VEL
LIN {X 0,Y 509.419,Z 692.672,A -85,B 0,C 180,E1 -5315.938,E2 -5315.938} C_VEL
LIN {X 0,Y 509.316,Z 698.014,A -85,B 0,C 180,E1 -5317.532,E2 -5317.532} C_VEL
LIN {X 0,Y 509.124,Z 703.129,A -85,B 0,C 180,E1 -5319.534,E2 -5319.534} C_VEL
LIN {X 0,Y 509.153,Z 706.021,A -85,B 0,C 180,E1 -5321.141,E2 -5321.141} C_VEL
LIN {X 0,Y 509.077,Z 707.937,A -85,B 0,C 180,E1 -5322.76,E2 -5322.76} C_VEL
LIN {X 0,Y 509.086,Z 708.846,A -85,B 0,C 180,E1 -5324.387,E2 -5324.387} C_VEL
LIN {X 0,Y 509.034,Z 708.755,A -85,B 0,C 180,E1 -5326.028,E2 -5326.028} C_VEL
LIN {X 0,Y 509.093,Z 707.608,A -85,B 0,C 180,E1 -5327.721,E2 -5327.721} C_VEL
LIN {X 0,Y 509.081,Z 705.458,A -85,B 0,C 180,E1 -5329.348,E2 -5329.348} C_VEL
LIN {X 0,Y 509.213,Z 701.014,A -85,B 0,C 180,E1 -5331.452,E2 -5331.452} C_VEL
LIN {X 0,Y 509.279,Z 697.473,A -85,B 0,C 180,E1 -5332.729,E2 -5332.729} C_VEL
LIN {X 0,Y 509.405,Z 693.243,A -85,B 0,C 180,E1 -5334.002,E2 -5334.002} C_VEL
LIN {X 0,Y 509.531,Z 688.081,A -85,B 0,C 180,E1 -5335.313,E2 -5335.313} C_VEL
LIN {X 0,Y 509.779,Z 680.859,A -85,B 0,C 180,E1 -5336.855,E2 -5336.855} C_VEL
LIN {X 0,Y 510.028,Z 673.941,A -85,B 0,C 180,E1 -5338.127,E2 -5338.127} C_VEL
LIN {X 0,Y 510.453,Z 665.4,A -85,B 0,C 180,E1 -5339.485,E2 -5339.485} C_VEL
LIN {X 0,Y 510.864,Z 657.435,A -85,B 0,C 180,E1 -5340.597,E2 -5340.597} C_VEL
LIN {X 0,Y 511.345,Z 648.556,A -85,B 0,C 180,E1 -5341.691,E2 -5341.691} C_VEL
LIN {X 0,Y 511.817,Z 639.092,A -85,B 0,C 180,E1 -5342.725,E2 -5342.725} C_VEL
LIN {X 0,Y 512.399,Z 628.456,A -85,B 0,C 180,E1 -5343.743,E2 -5343.743} C_VEL
LIN {X 0,Y 512.989,Z 617.905,A -85,B 0,C 180,E1 -5344.627,E2 -5344.627} C_VEL
LIN {X 0,Y 513.587,Z 606.806,A -85,B 0,C 180,E1 -5345.44,E2 -5345.44} C_VEL
LIN {X 0,Y 514.162,Z 595.598,A -85,B 0,C 180,E1 -5346.151,E2 -5346.151} C_VEL
LIN {X 0,Y 514.694,Z 583.275,A -85,B 0,C 180,E1 -5346.823,E2 -5346.823} C_VEL
LIN {X 0,Y 515.209,Z 571.245,A -85,B 0,C 180,E1 -5347.373,E2 -5347.373} C_VEL
LIN {X 0,Y 515.701,Z 557.803,A -85,B 0,C 180,E1 -5347.873,E2 -5347.873} C_VEL
LIN {X 0,Y 516.057,Z 543.318,A -85,B 0,C 180,E1 -5348.288,E2 -5348.288} C_VEL
LIN {X 0,Y 511.097,Z 527.148,A -85,B 0,C 180,E1 -5348.864,E2 -5348.864} C_VEL
LIN {X 0,Y 509.477,Z 522.328,A -85,B 0,C 180,E1 -5349.031,E2 -5349.031} C_VEL
LIN {X 0,Y 509.651,Z 517.82,A -85,B 0,C 180,E1 -5351.87,E2 -5351.87} C_VEL
LIN {X 0,Y 509.734,Z 512.976,A -85,B 0,C 180,E1 -5354.68,E2 -5354.68} C_VEL
LIN {X 0,Y 509.828,Z 508.086,A -85,B 0,C 180,E1 -5357.509,E2 -5357.509} C_VEL
LIN {X 0,Y 509.879,Z 502.504,A -85,B 0,C 180,E1 -5360.65,E2 -5360.65} C_VEL
LIN {X 0,Y 509.959,Z 496.91,A -85,B 0,C 180,E1 -5363.657,E2 -5363.657} C_VEL
LIN {X 0,Y 509.905,Z 495.285,A -85,B 0,C 180,E1 -5364.627,E2 -5364.627} C_VEL
LIN {X 0,Y 509.859,Z 495.291,A -85,B 0,C 180,E1 -5367.48,E2 -5367.48} C_VEL
LIN {X 0,Y 509.874,Z 495.288,A -85,B 0,C 180,E1 -5370.268,E2 -5370.268} C_VEL
LIN {X 0,Y 509.879,Z 495.286,A -85,B 0,C 180,E1 -5372.944,E2 -5372.944} C_VEL
LIN {X 0,Y 509.869,Z 495.287,A -85,B 0,C 180,E1 -5375.574,E2 -5375.574} C_VEL
LIN {X 0,Y 509.84,Z 495.291,A -85,B 0,C 180,E1 -5378.149,E2 -5378.149} C_VEL
LIN {X 0,Y 509.856,Z 495.288,A -85,B 0,C 180,E1 -5380.681,E2 -5380.681} C_VEL
LIN {X 0,Y 509.878,Z 495.285,A -85,B 0,C 180,E1 -5383.174,E2 -5383.174} C_VEL
LIN {X 0,Y 509.855,Z 495.29,A -85,B 0,C 180,E1 -5385.633,E2 -5385.633} C_VEL
LIN {X 0,Y 509.916,Z 495.278,A -85,B 0,C 180,E1 -5388.874,E2 -5388.874} C_VEL
LIN {X 0,Y 509.942,Z 495.275,A -85,B 0,C 180,E1 -5392.078,E2 -5392.078} C_VEL
LIN {X 0,Y 510.002,Z 495.268,A -85,B 0,C 180,E1 -5394.464,E2 -5394.464} C_VEL
LIN {X 0,Y 510.048,Z 495.265,A -85,B 0,C 180,E1 -5397.631,E2 -5397.631} C_VEL
LIN {X 0,Y 510.056,Z 495.264,A -85,B 0,C 180,E1 -5400.789,E2 -5400.789} C_VEL
LIN {X 0,Y 509.95,Z 495.276,A -85,B 0,C 180,E1 -5403.16,E2 -5403.16} C_VEL
LIN {X 0,Y 509.968,Z 495.275,A -85,B 0,C 180,E1 -5406.329,E2 -5406.329} C_VEL
LIN {X 0,Y 509.908,Z 495.28,A -85,B 0,C 180,E1 -5408.72,E2 -5408.72} C_VEL
LIN {X 0,Y 509.939,Z 495.274,A -85,B 0,C 180,E1 -5411.93,E2 -5411.93} C_VEL
LIN {X 0,Y 509.881,Z 495.284,A -85,B 0,C 180,E1 -5415.242,E2 -5415.242} C_VEL
LIN {X 0,Y 509.877,Z 495.268,A -85,B 0,C 180,E1 -5418.001,E2 -5418.001} C_VEL
LIN {X 0,Y 509.846,Z 495.292,A -85,B 0,C 180,E1 -5421.002,E2 -5421.002} C_VEL
LIN {X 0,Y 509.84,Z 495.282,A -85,B 0,C 180,E1 -5423.563,E2 -5423.563} C_VEL
LIN {X 0,Y 509.903,Z 495.279,A -85,B 0,C 180,E1 -5426.38,E2 -5426.38} C_VEL
LIN {X 0,Y 509.875,Z 495.286,A -85,B 0,C 180,E1 -5428.844,E2 -5428.844} C_VEL
LIN {X 0,Y 509.816,Z 495.294,A -85,B 0,C 180,E1 -5431.59,E2 -5431.59} C_VEL
LIN {X 0,Y 509.845,Z 495.291,A -85,B 0,C 180,E1 -5434.414,E2 -5434.414} C_VEL
LIN {X 0,Y 509.813,Z 495.295,A -85,B 0,C 180,E1 -5437.341,E2 -5437.341} C_VEL
LIN {X 0,Y 509.87,Z 495.286,A -85,B 0,C 180,E1 -5440.379,E2 -5440.379} C_VEL
LIN {X 0,Y 509.831,Z 495.293,A -85,B 0,C 180,E1 -5443.065,E2 -5443.065} C_VEL
LIN {X 0,Y 509.876,Z 495.392,A -85,B 0,C 180,E1 -5445.225,E2 -5445.225} C_VEL
LIN {X 0,Y 512.206,Z 505.989,A -85,B 0,C 180,E1 -5448.35,E2 -5448.35} C_VEL
LIN {X 0,Y 513.047,Z 509.881,A -85,B 0,C 180,E1 -5449.45,E2 -5449.45} C_VEL
LIN {X 0,Y 513.125,Z 517.052,A -85,B 0,C 180,E1 -5451.324,E2 -5451.324} C_VEL
LIN {X 0,Y 512.728,Z 529.307,A -85,B 0,C 180,E1 -5454.407,E2 -5454.407} C_VEL
LIN {X 0,Y 512.323,Z 540.865,A -85,B 0,C 180,E1 -5457.223,E2 -5457.223} C_VEL
LIN {X 0,Y 511.86,Z 552.659,A -85,B 0,C 180,E1 -5460.125,E2 -5460.125} C_VEL
LIN {X 0,Y 511.393,Z 564.57,A -85,B 0,C 180,E1 -5463.032,E2 -5463.032} C_VEL
LIN {X 0,Y 510.939,Z 577.14,A -85,B 0,C 180,E1 -5466.027,E2 -5466.027} C_VEL
LIN {X 0,Y 516.227,Z 596.408,A -85,B 0,C 180,E1 -5466.608,E2 -5466.608} C_VEL
LIN {X 0,Y 515.833,Z 613.768,A -85,B 0,C 180,E1 -5467.044,E2 -5467.044} C_VEL
LIN {X 0,Y 515.318,Z 629.57,A -85,B 0,C 180,E1 -5467.605,E2 -5467.605} C_VEL
LIN {X 0,Y 514.679,Z 644.123,A -85,B 0,C 180,E1 -5468.261,E2 -5468.261} C_VEL
LIN {X 0,Y 514.01,Z 658.732,A -85,B 0,C 180,E1 -5469.073,E2 -5469.073} C_VEL
LIN {X 0,Y 513.269,Z 673.696,A -85,B 0,C 180,E1 -5470.087,E2 -5470.087} C_VEL
LIN {X 0,Y 512.508,Z 686.458,A -85,B 0,C 180,E1 -5471.118,E2 -5471.118} C_VEL
LIN {X 0,Y 511.791,Z 700.078,A -85,B 0,C 180,E1 -5472.417,E2 -5472.417} C_VEL
LIN {X 0,Y 511.146,Z 712.643,A -85,B 0,C 180,E1 -5473.835,E2 -5473.835} C_VEL
LIN {X 0,Y 510.617,Z 723.345,A -85,B 0,C 180,E1 -5475.249,E2 -5475.249} C_VEL
LIN {X 0,Y 510.086,Z 733.677,A -85,B 0,C 180,E1 -5476.861,E2 -5476.861} C_VEL
LIN {X 0,Y 509.79,Z 742.49,A -85,B 0,C 180,E1 -5478.51,E2 -5478.51} C_VEL
LIN {X 0,Y 509.486,Z 749.494,A -85,B 0,C 180,E1 -5480.072,E2 -5480.072} C_VEL
LIN {X 0,Y 509.352,Z 755.469,A -85,B 0,C 180,E1 -5481.671,E2 -5481.671} C_VEL
LIN {X 0,Y 509.254,Z 761.25,A -85,B 0,C 180,E1 -5483.662,E2 -5483.662} C_VEL
LIN {X 0,Y 509.142,Z 764.637,A -85,B 0,C 180,E1 -5485.25,E2 -5485.25} C_VEL
LIN {X 0,Y 509.184,Z 767.091,A -85,B 0,C 180,E1 -5486.836,E2 -5486.836} C_VEL
LIN {X 0,Y 509.108,Z 768.48,A -85,B 0,C 180,E1 -5488.419,E2 -5488.419} C_VEL
LIN {X 0,Y 509.061,Z 769,A -85,B 0,C 180,E1 -5490.001,E2 -5490.001} C_VEL
LIN {X 0,Y 509.108,Z 768.479,A -85,B 0,C 180,E1 -5491.583,E2 -5491.583} C_VEL
LIN {X 0,Y 509.184,Z 767.088,A -85,B 0,C 180,E1 -5493.166,E2 -5493.166} C_VEL
LIN {X 0,Y 509.142,Z 764.634,A -85,B 0,C 180,E1 -5494.752,E2 -5494.752} C_VEL
LIN {X 0,Y 509.265,Z 760.878,A -85,B 0,C 180,E1 -5496.478,E2 -5496.478} C_VEL
LIN {X 0,Y 509.354,Z 755.465,A -85,B 0,C 180,E1 -5498.331,E2 -5498.331} C_VEL
LIN {X 0,Y 509.568,Z 747.853,A -85,B 0,C 180,E1 -5500.33,E2 -5500.33} C_VEL
LIN {X 0,Y 509.916,Z 739.249,A -85,B 0,C 180,E1 -5502.134,E2 -5502.134} C_VEL
LIN {X 0,Y 510.261,Z 729.972,A -85,B 0,C 180,E1 -5503.745,E2 -5503.745} C_VEL
LIN {X 0,Y 510.797,Z 719.221,A -85,B 0,C 180,E1 -5505.32,E2 -5505.32} C_VEL
LIN {X 0,Y 511.414,Z 707.499,A -85,B 0,C 180,E1 -5506.774,E2 -5506.774} C_VEL
LIN {X 0,Y 512.06,Z 695.037,A -85,B 0,C 180,E1 -5508.092,E2 -5508.092} C_VEL
LIN {X 0,Y 512.844,Z 681.459,A -85,B 0,C 180,E1 -5509.306,E2 -5509.306} C_VEL
LIN {X 0,Y 513.638,Z 666.558,A -85,B 0,C 180,E1 -5510.421,E2 -5510.421} C_VEL
LIN {X 0,Y 514.396,Z 651.736,A -85,B 0,C 180,E1 -5511.332,E2 -5511.332} C_VEL
LIN {X 0,Y 515.035,Z 636.635,A -85,B 0,C 180,E1 -5512.093,E2 -5512.093} C_VEL
LIN {X 0,Y 515.692,Z 619.872,A -85,B 0,C 180,E1 -5512.753,E2 -5512.753} C_VEL
LIN {X 0,Y 516.11,Z 603.532,A -85,B 0,C 180,E1 -5513.232,E2 -5513.232} C_VEL
LIN {X 0,Y 516.096,Z 595.95,A -85,B 0,C 180,E1 -5513.409,E2 -5513.409} C_VEL
LIN {X 0,Y 510.927,Z 577.115,A -85,B 0,C 180,E1 -5513.979,E2 -5513.979} C_VEL
LIN {X 0,Y 511.396,Z 564.562,A -85,B 0,C 180,E1 -5516.97,E2 -5516.97} C_VEL
LIN {X 0,Y 511.91,Z 551.638,A -85,B 0,C 180,E1 -5520.127,E2 -5520.127} C_VEL
LIN {X 0,Y 512.244,Z 542.652,A -85,B 0,C 180,E1 -5522.35,E2 -5522.35} C_VEL
LIN {X 0,Y 512.402,Z 529.452,A -85,B 0,C 180,E1 -5525.175,E2 -5525.175} C_VEL
LIN {X 0,Y 512.363,Z 516.859,A -85,B 0,C 180,E1 -5527.891,E2 -5527.891} C_VEL
LIN {X 0,Y 512.321,Z 508.263,A -85,B 0,C 180,E1 -5529.807,E2 -5529.807} C_VEL
LIN {X 0,Y 510.915,Z 500.729,A -85,B 0,C 180,E1 -5531.644,E2 -5531.644} C_VEL
LIN {X 0,Y 509.861,Z 495.291,A -85,B 0,C 180,E1 -5533.107,E2 -5533.107} C_VEL
LIN {X 0,Y 509.832,Z 495.29,A -85,B 0,C 180,E1 -5535.793,E2 -5535.793} C_VEL
LIN {X 0,Y 509.858,Z 495.291,A -85,B 0,C 180,E1 -5538.575,E2 -5538.575} C_VEL
LIN {X 0,Y 509.852,Z 495.288,A -85,B 0,C 180,E1 -5541.787,E2 -5541.787} C_VEL
LIN {X 0,Y 509.844,Z 495.292,A -85,B 0,C 180,E1 -5544.623,E2 -5544.623} C_VEL
LIN {X 0,Y 509.864,Z 495.286,A -85,B 0,C 180,E1 -5547.481,E2 -5547.481} C_VEL
LIN {X 0,Y 509.86,Z 495.29,A -85,B 0,C 180,E1 -5550.274,E2 -5550.274} C_VEL
LIN {X 0,Y 509.887,Z 495.283,A -85,B 0,C 180,E1 -5552.945,E2 -5552.945} C_VEL
LIN {X 0,Y 509.891,Z 495.287,A -85,B 0,C 180,E1 -5556.008,E2 -5556.008} C_VEL
LIN {X 0,Y 509.886,Z 495.286,A -85,B 0,C 180,E1 -5556.374,E2 -5556.374} C_VEL
LIN {X 0,Y 511.627,Z 500.155,A -85,B 0,C 180,E1 -5556.552,E2 -5556.552} C_VEL
LIN {X 0,Y 515.911,Z 510.644,A -85,B 0,C 180,E1 -5557.016,E2 -5557.016} C_VEL
LIN {X 0,Y 515.477,Z 525.288,A -85,B 0,C 180,E1 -5557.489,E2 -5557.489} C_VEL
LIN {X 0,Y 514.869,Z 541.131,A -85,B 0,C 180,E1 -5558.157,E2 -5558.157} C_VEL
LIN {X 0,Y 514.14,Z 556.354,A -85,B 0,C 180,E1 -5558.972,E2 -5558.972} C_VEL
LIN {X 0,Y 513.361,Z 571.668,A -85,B 0,C 180,E1 -5559.986,E2 -5559.986} C_VEL
LIN {X 0,Y 512.572,Z 585.736,A -85,B 0,C 180,E1 -5561.099,E2 -5561.099} C_VEL
LIN {X 0,Y 511.929,Z 598.716,A -85,B 0,C 180,E1 -5562.318,E2 -5562.318} C_VEL
LIN {X 0,Y 511.234,Z 610.641,A -85,B 0,C 180,E1 -5563.632,E2 -5563.632} C_VEL
LIN {X 0,Y 510.743,Z 621.591,A -85,B 0,C 180,E1 -5565.049,E2 -5565.049} C_VEL
LIN {X 0,Y 510.16,Z 632.181,A -85,B 0,C 180,E1 -5566.659,E2 -5566.659} C_VEL
LIN {X 0,Y 509.886,Z 640.377,A -85,B 0,C 180,E1 -5568.133,E2 -5568.133} C_VEL
LIN {X 0,Y 509.574,Z 647.638,A -85,B 0,C 180,E1 -5569.672,E2 -5569.672} C_VEL
LIN {X 0,Y 509.407,Z 653.905,A -85,B 0,C 180,E1 -5571.271,E2 -5571.271} C_VEL
LIN {X 0,Y 509.31,Z 658.996,A -85,B 0,C 180,E1 -5572.866,E2 -5572.866} C_VEL
LIN {X 0,Y 509.217,Z 662.972,A -85,B 0,C 180,E1 -5574.456,E2 -5574.456} C_VEL
LIN {X 0,Y 509.196,Z 665.917,A -85,B 0,C 180,E1 -5576.043,E2 -5576.043} C_VEL
LIN {X 0,Y 509.154,Z 667.875,A -85,B 0,C 180,E1 -5577.627,E2 -5577.627} C_VEL
LIN {X 0,Y 509.071,Z 668.861,A -85,B 0,C 180,E1 -5579.209,E2 -5579.209} C_VEL
LIN {X 0,Y 509.071,Z 668.877,A -85,B 0,C 180,E1 -5580.791,E2 -5580.791} C_VEL
LIN {X 0,Y 509.154,Z 667.945,A -85,B 0,C 180,E1 -5582.374,E2 -5582.374} C_VEL
LIN {X 0,Y 509.198,Z 666.05,A -85,B 0,C 180,E1 -5583.958,E2 -5583.958} C_VEL
LIN {X 0,Y 509.218,Z 663.164,A -85,B 0,C 180,E1 -5585.544,E2 -5585.544} C_VEL
LIN {X 0,Y 509.311,Z 659.259,A -85,B 0,C 180,E1 -5587.134,E2 -5587.134} C_VEL
LIN {X 0,Y 509.403,Z 654.24,A -85,B 0,C 180,E1 -5588.729,E2 -5588.729} C_VEL
LIN {X 0,Y 509.564,Z 648.047,A -85,B 0,C 180,E1 -5590.329,E2 -5590.329} C_VEL
LIN {X 0,Y 509.843,Z 640.528,A -85,B 0,C 180,E1 -5591.933,E2 -5591.933} C_VEL
LIN {X 0,Y 510.202,Z 631.506,A -85,B 0,C 180,E1 -5593.543,E2 -5593.543} C_VEL
LIN {X 0,Y 510.771,Z 620.757,A -85,B 0,C 180,E1 -5595.155,E2 -5595.155} C_VEL
LIN {X 0,Y 511.275,Z 609.65,A -85,B 0,C 180,E1 -5596.573,E2 -5596.573} C_VEL
LIN {X 0,Y 511.89,Z 598.54,A -85,B 0,C 180,E1 -5597.788,E2 -5597.788} C_VEL
LIN {X 0,Y 512.668,Z 585.037,A -85,B 0,C 180,E1 -5599.049,E2 -5599.049} C_VEL
LIN {X 0,Y 513.375,Z 571.508,A -85,B 0,C 180,E1 -5600.118,E2 -5600.118} C_VEL
LIN {X 0,Y 514.105,Z 557.801,A -85,B 0,C 180,E1 -5601.03,E2 -5601.03} C_VEL
LIN {X 0,Y 514.834,Z 541.985,A -85,B 0,C 180,E1 -5601.891,E2 -5601.891} C_VEL
LIN {X 0,Y 515.417,Z 527.209,A -85,B 0,C 180,E1 -5602.529,E2 -5602.529} C_VEL
LIN {X 0,Y 515.783,Z 509.901,A -85,B 0,C 180,E1 -5603.111,E2 -5603.111} C_VEL
LIN {X 0,Y 509.97,Z 495.885,A -85,B 0,C 180,E1 -5603.726,E2 -5603.726} C_VEL
LIN {X 0,Y 509.877,Z 495.287,A -85,B 0,C 180,E1 -5603.777,E2 -5603.777} C_VEL
LIN {X 0,Y 509.915,Z 495.282,A -85,B 0,C 180,E1 -5606.379,E2 -5606.379} C_VEL
LIN {X 0,Y 509.88,Z 495.288,A -85,B 0,C 180,E1 -5608.844,E2 -5608.844} C_VEL
LIN {X 0,Y 509.824,Z 495.295,A -85,B 0,C 180,E1 -5611.59,E2 -5611.59} C_VEL
LIN {X 0,Y 509.857,Z 495.29,A -85,B 0,C 180,E1 -5614.413,E2 -5614.413} C_VEL
LIN {X 0,Y 509.823,Z 495.294,A -85,B 0,C 180,E1 -5617.341,E2 -5617.341} C_VEL
LIN {X 0,Y 509.843,Z 495.293,A -85,B 0,C 180,E1 -5620.382,E2 -5620.382} C_VEL
LIN {X 0,Y 509.828,Z 495.294,A -85,B 0,C 180,E1 -5623.062,E2 -5623.062} C_VEL
LIN {X 0,Y 509.843,Z 495.292,A -85,B 0,C 180,E1 -5624.692,E2 -5624.692} C_VEL
LIN {X 0,Y 509.162,Z 495.374,A -85,B 0,C 180,E1 -5625.351,E2 -5625.351} C_VEL
LIN {X 0,Y 506.308,Z 495.73,A -85,B 0,C 180,E1 -5626.421,E2 -5626.421} C_VEL
LIN {X 0,Y 503.905,Z 496.031,A -85,B 0,C 180,E1 -5627.284,E2 -5627.284} C_VEL
LIN {X 0,Y 502.875,Z 496.157,A -85,B 0,C 180,E1 -5627.949,E2 -5627.949} C_VEL
LIN {X 0,Y 502.792,Z 496.167,A -85,B 0,C 180,E1 -5628.175,E2 -5628.175} C_VEL
LIN {X 0,Y 502.807,Z 496.166,A -85,B 0,C 180,E1 -5631.024,E2 -5631.024} C_VEL
LIN {X 0,Y 502.78,Z 496.171,A -85,B 0,C 180,E1 -5634.169,E2 -5634.169} C_VEL
LIN {X 0,Y 502.838,Z 496.164,A -85,B 0,C 180,E1 -5636.993,E2 -5636.993} C_VEL
LIN {X 0,Y 502.821,Z 496.168,A -85,B 0,C 180,E1 -5640.065,E2 -5640.065} C_VEL
LIN {X 0,Y 502.838,Z 496.163,A -85,B 0,C 180,E1 -5642.533,E2 -5642.533} C_VEL
LIN {X 0,Y 502.94,Z 496.269,A -85,B 0,C 180,E1 -5645.486,E2 -5645.486} C_VEL
LIN {X 0,Y 502.872,Z 502.158,A -85,B 0,C 180,E1 -5648.692,E2 -5648.692} C_VEL
LIN {X 0,Y 502.83,Z 506.725,A -85,B 0,C 180,E1 -5651.248,E2 -5651.248} C_VEL
LIN {X 0,Y 502.769,Z 511.073,A -85,B 0,C 180,E1 -5653.765,E2 -5653.765} C_VEL
LIN {X 0,Y 502.699,Z 515.309,A -85,B 0,C 180,E1 -5656.25,E2 -5656.25} C_VEL
LIN {X 0,Y 502.688,Z 519.395,A -85,B 0,C 180,E1 -5658.712,E2 -5658.712} C_VEL
LIN {X 0,Y 502.534,Z 522.723,A -85,B 0,C 180,E1 -5660.718,E2 -5660.718} C_VEL
LIN {X 0,Y 505.053,Z 529.87,A -85,B 0,C 180,E1 -5660.964,E2 -5660.964} C_VEL
LIN {X 0,Y 509.592,Z 544.823,A -85,B 0,C 180,E1 -5661.521,E2 -5661.521} C_VEL
LIN {X 0,Y 509.103,Z 561.218,A -85,B 0,C 180,E1 -5662.012,E2 -5662.012} C_VEL
LIN {X 0,Y 508.463,Z 577.186,A -85,B 0,C 180,E1 -5662.654,E2 -5662.654} C_VEL
LIN {X 0,Y 507.746,Z 592.464,A -85,B 0,C 180,E1 -5663.442,E2 -5663.442} C_VEL
LIN {X 0,Y 507.057,Z 605.094,A -85,B 0,C 180,E1 -5664.232,E2 -5664.232} C_VEL
LIN {X 0,Y 506.342,Z 617.184,A -85,B 0,C 180,E1 -5665.122,E2 -5665.122} C_VEL
LIN {X 0,Y 505.693,Z 627.684,A -85,B 0,C 180,E1 -5666.015,E2 -5666.015} C_VEL
LIN {X 0,Y 505.061,Z 638.009,A -85,B 0,C 180,E1 -5667.008,E2 -5667.008} C_VEL
LIN {X 0,Y 504.509,Z 647.174,A -85,B 0,C 180,E1 -5668.003,E2 -5668.003} C_VEL
LIN {X 0,Y 504.039,Z 655.355,A -85,B 0,C 180,E1 -5669,E2 -5669} C_VEL
LIN {X 0,Y 503.519,Z 664.054,A -85,B 0,C 180,E1 -5670.199,E2 -5670.199} C_VEL
LIN {X 0,Y 503.133,Z 671.719,A -85,B 0,C 180,E1 -5671.4,E2 -5671.4} C_VEL
LIN {X 0,Y 502.84,Z 678.479,A -85,B 0,C 180,E1 -5672.603,E2 -5672.603} C_VEL
LIN {X 0,Y 502.59,Z 685.324,A -85,B 0,C 180,E1 -5674.008,E2 -5674.008} C_VEL
LIN {X 0,Y 502.369,Z 690.441,A -85,B 0,C 180,E1 -5675.216,E2 -5675.216} C_VEL
LIN {X 0,Y 502.243,Z 696.145,A -85,B 0,C 180,E1 -5676.83,E2 -5676.83} C_VEL
LIN {X 0,Y 502.212,Z 699.73,A -85,B 0,C 180,E1 -5678.043,E2 -5678.043} C_VEL
LIN {X 0,Y 502.035,Z 703.542,A -85,B 0,C 180,E1 -5679.67,E2 -5679.67} C_VEL
LIN {X 0,Y 502.064,Z 706.316,A -85,B 0,C 180,E1 -5681.301,E2 -5681.301} C_VEL
LIN {X 0,Y 502.018,Z 707.408,A -85,B 0,C 180,E1 -5682.121,E2 -5682.121} C_VEL
LIN {X 0,Y 501.99,Z 708.673,A -85,B 0,C 180,E1 -5683.768,E2 -5683.768} C_VEL
LIN {X 0,Y 501.939,Z 708.92,A -85,B 0,C 180,E1 -5685.427,E2 -5685.427} C_VEL
LIN {X 0,Y 501.986,Z 708.152,A -85,B 0,C 180,E1 -5687.097,E2 -5687.097} C_VEL
LIN {X 0,Y 501.989,Z 707.438,A -85,B 0,C 180,E1 -5687.938,E2 -5687.938} C_VEL
LIN {X 0,Y 502.017,Z 705.075,A -85,B 0,C 180,E1 -5689.631,E2 -5689.631} C_VEL
LIN {X 0,Y 502.142,Z 700.434,A -85,B 0,C 180,E1 -5691.77,E2 -5691.77} C_VEL
LIN {X 0,Y 502.204,Z 696.749,A -85,B 0,C 180,E1 -5693.068,E2 -5693.068} C_VEL
LIN {X 0,Y 502.366,Z 691.524,A -85,B 0,C 180,E1 -5694.585,E2 -5694.585} C_VEL
LIN {X 0,Y 502.506,Z 687.045,A -85,B 0,C 180,E1 -5695.693,E2 -5695.693} C_VEL
LIN {X 0,Y 502.773,Z 680.873,A -85,B 0,C 180,E1 -5697.019,E2 -5697.019} C_VEL
LIN {X 0,Y 503.06,Z 673.666,A -85,B 0,C 180,E1 -5698.358,E2 -5698.358} C_VEL
LIN {X 0,Y 503.503,Z 665.304,A -85,B 0,C 180,E1 -5699.702,E2 -5699.702} C_VEL
LIN {X 0,Y 503.945,Z 657.321,A -85,B 0,C 180,E1 -5700.83,E2 -5700.83} C_VEL
LIN {X 0,Y 504.484,Z 648.234,A -85,B 0,C 180,E1 -5701.962,E2 -5701.962} C_VEL
LIN {X 0,Y 505.029,Z 638.366,A -85,B 0,C 180,E1 -5703.046,E2 -5703.046} C_VEL
LIN {X 0,Y 505.7,Z 627.094,A -85,B 0,C 180,E1 -5704.131,E2 -5704.131} C_VEL
LIN {X 0,Y 506.6,Z 613.438,A -85,B 0,C 180,E1 -5705.267,E2 -5705.267} C_VEL
LIN {X 0,Y 507.435,Z 598.26,A -85,B 0,C 180,E1 -5706.304,E2 -5706.304} C_VEL
LIN {X 0,Y 508.093,Z 584.652,A -85,B 0,C 180,E1 -5707.077,E2 -5707.077} C_VEL
LIN {X 0,Y 508.773,Z 569.434,A -85,B 0,C 180,E1 -5707.771,E2 -5707.771} C_VEL
LIN {X 0,Y 509.382,Z 552.635,A -85,B 0,C 180,E1 -5708.358,E2 -5708.358} C_VEL
LIN {X 0,Y 509.424,Z 544.297,A -85,B 0,C 180,E1 -5708.592,E2 -5708.592} C_VEL
LIN {X 0,Y 504.558,Z 528.596,A -85,B 0,C 180,E1 -5709.173,E2 -5709.173} C_VEL
LIN {X 0,Y 502.447,Z 522.749,A -85,B 0,C 180,E1 -5709.393,E2 -5709.393} C_VEL
LIN {X 0,Y 502.62,Z 518.247,A -85,B 0,C 180,E1 -5712.175,E2 -5712.175} C_VEL
LIN {X 0,Y 502.75,Z 512.663,A -85,B 0,C 180,E1 -5715.472,E2 -5715.472} C_VEL
LIN {X 0,Y 502.824,Z 508.482,A -85,B 0,C 180,E1 -5717.863,E2 -5717.863} C_VEL
LIN {X 0,Y 502.847,Z 504.333,A -85,B 0,C 180,E1 -5720.235,E2 -5720.235} C_VEL
LIN {X 0,Y 502.887,Z 499.158,A -85,B 0,C 180,E1 -5723.062,E2 -5723.062} C_VEL
LIN {X 0,Y 502.859,Z 496.163,A -85,B 0,C 180,E1 -5724.7,E2 -5724.7} C_VEL
LIN {X 0,Y 502.781,Z 496.175,A -85,B 0,C 180,E1 -5727.915,E2 -5727.915} C_VEL
LIN {X 0,Y 502.831,Z 496.166,A -85,B 0,C 180,E1 -5730.712,E2 -5730.712} C_VEL
LIN {X 0,Y 502.872,Z 496.16,A -85,B 0,C 180,E1 -5733.434,E2 -5733.434} C_VEL
LIN {X 0,Y 502.795,Z 496.171,A -85,B 0,C 180,E1 -5736.086,E2 -5736.086} C_VEL
LIN {X 0,Y 502.788,Z 496.171,A -85,B 0,C 180,E1 -5738.689,E2 -5738.689} C_VEL
LIN {X 0,Y 502.836,Z 496.165,A -85,B 0,C 180,E1 -5741.877,E2 -5741.877} C_VEL
LIN {X 0,Y 502.829,Z 496.165,A -85,B 0,C 180,E1 -5744.662,E2 -5744.662} C_VEL
LIN {X 0,Y 502.889,Z 496.157,A -85,B 0,C 180,E1 -5748.026,E2 -5748.026} C_VEL
LIN {X 0,Y 502.868,Z 496.16,A -85,B 0,C 180,E1 -5751.156,E2 -5751.156} C_VEL
LIN {X 0,Y 502.922,Z 496.153,A -85,B 0,C 180,E1 -5753.581,E2 -5753.581} C_VEL
LIN {X 0,Y 502.894,Z 496.157,A -85,B 0,C 180,E1 -5756.795,E2 -5756.795} C_VEL
LIN {X 0,Y 503.027,Z 496.138,A -85,B 0,C 180,E1 -5759.199,E2 -5759.199} C_VEL
LIN {X 0,Y 502.893,Z 496.154,A -85,B 0,C 180,E1 -5761.601,E2 -5761.601} C_VEL
LIN {X 0,Y 502.894,Z 496.156,A -85,B 0,C 180,E1 -5763.204,E2 -5763.204} C_VEL
LIN {X 0,Y 502.917,Z 496.152,A -85,B 0,C 180,E1 -5766.418,E2 -5766.418} C_VEL
LIN {X 0,Y 502.867,Z 496.156,A -85,B 0,C 180,E1 -5768.843,E2 -5768.843} C_VEL
LIN {X 0,Y 502.882,Z 496.152,A -85,B 0,C 180,E1 -5772.1,E2 -5772.1} C_VEL
LIN {X 0,Y 502.836,Z 496.163,A -85,B 0,C 180,E1 -5775.4,E2 -5775.4} C_VEL
LIN {X 0,Y 502.834,Z 496.145,A -85,B 0,C 180,E1 -5778.123,E2 -5778.123} C_VEL
LIN {X 0,Y 502.786,Z 496.17,A -85,B 0,C 180,E1 -5781.311,E2 -5781.311} C_VEL
LIN {X 0,Y 502.791,Z 496.154,A -85,B 0,C 180,E1 -5783.913,E2 -5783.913} C_VEL
LIN {X 0,Y 502.87,Z 496.157,A -85,B 0,C 180,E1 -5786.565,E2 -5786.565} C_VEL
LIN {X 0,Y 502.828,Z 496.166,A -85,B 0,C 180,E1 -5789.287,E2 -5789.287} C_VEL
LIN {X 0,Y 502.778,Z 496.172,A -85,B 0,C 180,E1 -5792.085,E2 -5792.085} C_VEL
LIN {X 0,Y 502.8,Z 496.167,A -85,B 0,C 180,E1 -5794.965,E2 -5794.965} C_VEL
LIN {X 0,Y 502.789,Z 496.167,A -85,B 0,C 180,E1 -5797.954,E2 -5797.954} C_VEL
LIN {X 0,Y 502.822,Z 496.164,A -85,B 0,C 180,E1 -5801.065,E2 -5801.065} C_VEL
LIN {X 0,Y 502.773,Z 496.172,A -85,B 0,C 180,E1 -5803.376,E2 -5803.376} C_VEL
LIN {X 0,Y 502.839,Z 496.347,A -85,B 0,C 180,E1 -5804.835,E2 -5804.835} C_VEL
LIN {X 0,Y 504.838,Z 505.282,A -85,B 0,C 180,E1 -5807.546,E2 -5807.546} C_VEL
LIN {X 0,Y 506.109,Z 511.22,A -85,B 0,C 180,E1 -5809.259,E2 -5809.259} C_VEL
LIN {X 0,Y 506.317,Z 517.789,A -85,B 0,C 180,E1 -5811.015,E2 -5811.015} C_VEL
LIN {X 0,Y 505.812,Z 530.621,A -85,B 0,C 180,E1 -5814.3,E2 -5814.3} C_VEL
LIN {X 0,Y 505.377,Z 542.187,A -85,B 0,C 180,E1 -5817.158,E2 -5817.158} C_VEL
LIN {X 0,Y 504.972,Z 553.673,A -85,B 0,C 180,E1 -5819.933,E2 -5819.933} C_VEL
LIN {X 0,Y 504.515,Z 564.57,A -85,B 0,C 180,E1 -5822.634,E2 -5822.634} C_VEL
LIN {X 0,Y 503.98,Z 577.103,A -85,B 0,C 180,E1 -5825.666,E2 -5825.666} C_VEL
LIN {X 0,Y 509.702,Z 597.82,A -85,B 0,C 180,E1 -5826.323,E2 -5826.323} C_VEL
LIN {X 0,Y 509.293,Z 614.333,A -85,B 0,C 180,E1 -5826.75,E2 -5826.75} C_VEL
LIN {X 0,Y 508.708,Z 630.866,A -85,B 0,C 180,E1 -5827.351,E2 -5827.351} C_VEL
LIN {X 0,Y 507.987,Z 646.105,A -85,B 0,C 180,E1 -5828.067,E2 -5828.067} C_VEL
LIN {X 0,Y 507.155,Z 661.894,A -85,B 0,C 180,E1 -5828.989,E2 -5828.989} C_VEL
LIN {X 0,Y 506.391,Z 676.336,A -85,B 0,C 180,E1 -5830.017,E2 -5830.017} C_VEL
LIN {X 0,Y 505.604,Z 689.195,A -85,B 0,C 180,E1 -5831.098,E2 -5831.098} C_VEL
LIN {X 0,Y 504.84,Z 702.025,A -85,B 0,C 180,E1 -5832.376,E2 -5832.376} C_VEL
LIN {X 0,Y 504.151,Z 714.269,A -85,B 0,C 180,E1 -5833.812,E2 -5833.812} C_VEL
LIN {X 0,Y 503.572,Z 724.707,A -85,B 0,C 180,E1 -5835.245,E2 -5835.245} C_VEL
LIN {X 0,Y 503.038,Z 734.82,A -85,B 0,C 180,E1 -5836.879,E2 -5836.879} C_VEL
LIN {X 0,Y 502.734,Z 743.14,A -85,B 0,C 180,E1 -5838.479,E2 -5838.479} C_VEL
LIN {X 0,Y 502.431,Z 749.494,A -85,B 0,C 180,E1 -5839.931,E2 -5839.931} C_VEL
LIN {X 0,Y 502.297,Z 755.469,A -85,B 0,C 180,E1 -5841.553,E2 -5841.553} C_VEL
LIN {X 0,Y 502.182,Z 761.251,A -85,B 0,C 180,E1 -5843.573,E2 -5843.573} C_VEL
LIN {X 0,Y 502.061,Z 764.637,A -85,B 0,C 180,E1 -5845.183,E2 -5845.183} C_VEL
LIN {X 0,Y 502.102,Z 767.091,A -85,B 0,C 180,E1 -5846.791,E2 -5846.791} C_VEL
LIN {X 0,Y 502.031,Z 768.48,A -85,B 0,C 180,E1 -5848.396,E2 -5848.396} C_VEL
LIN {X 0,Y 501.975,Z 769,A -85,B 0,C 180,E1 -5850.001,E2 -5850.001} C_VEL
LIN {X 0,Y 502.031,Z 768.478,A -85,B 0,C 180,E1 -5851.605,E2 -5851.605} C_VEL
LIN {X 0,Y 502.103,Z 767.088,A -85,B 0,C 180,E1 -5853.21,E2 -5853.21} C_VEL
LIN {X 0,Y 502.061,Z 764.633,A -85,B 0,C 180,E1 -5854.819,E2 -5854.819} C_VEL
LIN {X 0,Y 502.183,Z 761.141,A -85,B 0,C 180,E1 -5856.47,E2 -5856.47} C_VEL
LIN {X 0,Y 502.299,Z 755.465,A -85,B 0,C 180,E1 -5858.449,E2 -5858.449} C_VEL
LIN {X 0,Y 502.511,Z 747.853,A -85,B 0,C 180,E1 -5860.476,E2 -5860.476} C_VEL
LIN {X 0,Y 502.881,Z 739.25,A -85,B 0,C 180,E1 -5862.306,E2 -5862.306} C_VEL
LIN {X 0,Y 503.28,Z 729.972,A -85,B 0,C 180,E1 -5863.94,E2 -5863.94} C_VEL
LIN {X 0,Y 503.813,Z 720.417,A -85,B 0,C 180,E1 -5865.37,E2 -5865.37} C_VEL
LIN {X 0,Y 504.415,Z 709.277,A -85,B 0,C 180,E1 -5866.805,E2 -5866.805} C_VEL
LIN {X 0,Y 505.138,Z 697.134,A -85,B 0,C 180,E1 -5868.138,E2 -5868.138} C_VEL
LIN {X 0,Y 505.943,Z 683.768,A -85,B 0,C 180,E1 -5869.378,E2 -5869.378} C_VEL
LIN {X 0,Y 506.778,Z 669.412,A -85,B 0,C 180,E1 -5870.498,E2 -5870.498} C_VEL
LIN {X 0,Y 507.538,Z 655.407,A -85,B 0,C 180,E1 -5871.413,E2 -5871.413} C_VEL
LIN {X 0,Y 508.322,Z 640.231,A -85,B 0,C 180,E1 -5872.229,E2 -5872.229} C_VEL
LIN {X 0,Y 508.958,Z 624.974,A -85,B 0,C 180,E1 -5872.88,E2 -5872.88} C_VEL
LIN {X 0,Y 509.436,Z 608.737,A -85,B 0,C 180,E1 -5873.41,E2 -5873.41} C_VEL
LIN {X 0,Y 509.574,Z 597.311,A -85,B 0,C 180,E1 -5873.695,E2 -5873.695} C_VEL
LIN {X 0,Y 503.988,Z 577.089,A -85,B 0,C 180,E1 -5874.337,E2 -5874.337} C_VEL
LIN {X 0,Y 504.443,Z 566.403,A -85,B 0,C 180,E1 -5876.918,E2 -5876.918} C_VEL
LIN {X 0,Y 504.916,Z 555.481,A -85,B 0,C 180,E1 -5879.613,E2 -5879.613} C_VEL
LIN {X 0,Y 505.168,Z 547.85,A -85,B 0,C 180,E1 -5881.447,E2 -5881.447} C_VEL
LIN {X 0,Y 505.281,Z 535.781,A -85,B 0,C 180,E1 -5884.045,E2 -5884.045} C_VEL
LIN {X 0,Y 505.413,Z 523.458,A -85,B 0,C 180,E1 -5886.723,E2 -5886.723} C_VEL
LIN {X 0,Y 505.391,Z 511.017,A -85,B 0,C 180,E1 -5889.521,E2 -5889.521} C_VEL
LIN {X 0,Y 504.951,Z 506.747,A -85,B 0,C 180,E1 -5890.547,E2 -5890.547} C_VEL
LIN {X 0,Y 502.859,Z 496.441,A -85,B 0,C 180,E1 -5893.298,E2 -5893.298} C_VEL
LIN {X 0,Y 502.8,Z 496.17,A -85,B 0,C 180,E1 -5893.378,E2 -5893.378} C_VEL
LIN {X 0,Y 502.783,Z 496.172,A -85,B 0,C 180,E1 -5896.625,E2 -5896.625} C_VEL
LIN {X 0,Y 502.82,Z 496.166,A -85,B 0,C 180,E1 -5899.006,E2 -5899.006} C_VEL
LIN {X 0,Y 502.795,Z 496.169,A -85,B 0,C 180,E1 -5902.047,E2 -5902.047} C_VEL
LIN {X 0,Y 502.809,Z 496.166,A -85,B 0,C 180,E1 -5905.035,E2 -5905.035} C_VEL
LIN {X 0,Y 502.786,Z 496.17,A -85,B 0,C 180,E1 -5907.916,E2 -5907.916} C_VEL
LIN {X 0,Y 502.826,Z 496.164,A -85,B 0,C 180,E1 -5910.713,E2 -5910.713} C_VEL
LIN {X 0,Y 502.864,Z 496.159,A -85,B 0,C 180,E1 -5913.44,E2 -5913.44} C_VEL
LIN {X 0,Y 502.851,Z 496.164,A -85,B 0,C 180,E1 -5916.062,E2 -5916.062} C_VEL
LIN {X 0,Y 504.727,Z 501.226,A -85,B 0,C 180,E1 -5916.264,E2 -5916.264} C_VEL
LIN {X 0,Y 509.26,Z 512.398,A -85,B 0,C 180,E1 -5916.77,E2 -5916.77} C_VEL
LIN {X 0,Y 508.769,Z 528.176,A -85,B 0,C 180,E1 -5917.299,E2 -5917.299} C_VEL
LIN {X 0,Y 508.075,Z 544.264,A -85,B 0,C 180,E1 -5918.011,E2 -5918.011} C_VEL
LIN {X 0,Y 507.331,Z 559.9,A -85,B 0,C 180,E1 -5918.889,E2 -5918.889} C_VEL
LIN {X 0,Y 506.526,Z 574.776,A -85,B 0,C 180,E1 -5919.916,E2 -5919.916} C_VEL
LIN {X 0,Y 505.676,Z 588.771,A -85,B 0,C 180,E1 -5921.084,E2 -5921.084} C_VEL
LIN {X 0,Y 504.871,Z 601.688,A -85,B 0,C 180,E1 -5922.376,E2 -5922.376} C_VEL
LIN {X 0,Y 504.155,Z 613.941,A -85,B 0,C 180,E1 -5923.812,E2 -5923.812} C_VEL
LIN {X 0,Y 503.589,Z 624.434,A -85,B 0,C 180,E1 -5925.245,E2 -5925.245} C_VEL
LIN {X 0,Y 503.052,Z 634.576,A -85,B 0,C 180,E1 -5926.878,E2 -5926.878} C_VEL
LIN {X 0,Y 502.743,Z 642.894,A -85,B 0,C 180,E1 -5928.473,E2 -5928.473} C_VEL
LIN {X 0,Y 502.361,Z 650.931,A -85,B 0,C 180,E1 -5930.336,E2 -5930.336} C_VEL
LIN {X 0,Y 502.249,Z 656.596,A -85,B 0,C 180,E1 -5931.957,E2 -5931.957} C_VEL
LIN {X 0,Y 502.186,Z 661.119,A -85,B 0,C 180,E1 -5933.572,E2 -5933.572} C_VEL
LIN {X 0,Y 502.063,Z 664.567,A -85,B 0,C 180,E1 -5935.182,E2 -5935.182} C_VEL
LIN {X 0,Y 502.106,Z 667.017,A -85,B 0,C 180,E1 -5936.791,E2 -5936.791} C_VEL
LIN {X 0,Y 502.03,Z 668.486,A -85,B 0,C 180,E1 -5938.396,E2 -5938.396} C_VEL
LIN {X 0,Y 501.978,Z 668.997,A -85,B 0,C 180,E1 -5940,E2 -5940} C_VEL
LIN {X 0,Y 502.03,Z 668.53,A -85,B 0,C 180,E1 -5941.605,E2 -5941.605} C_VEL
LIN {X 0,Y 502.107,Z 667.117,A -85,B 0,C 180,E1 -5943.21,E2 -5943.21} C_VEL
LIN {X 0,Y 502.063,Z 664.73,A -85,B 0,C 180,E1 -5944.818,E2 -5944.818} C_VEL
LIN {X 0,Y 502.189,Z 660.821,A -85,B 0,C 180,E1 -5946.631,E2 -5946.631} C_VEL
LIN {X 0,Y 502.286,Z 655.582,A -85,B 0,C 180,E1 -5948.449,E2 -5948.449} C_VEL
LIN {X 0,Y 502.428,Z 649.677,A -85,B 0,C 180,E1 -5950.07,E2 -5950.07} C_VEL
LIN {X 0,Y 502.807,Z 641.418,A -85,B 0,C 180,E1 -5951.922,E2 -5951.922} C_VEL
LIN {X 0,Y 503.141,Z 632.74,A -85,B 0,C 180,E1 -5953.531,E2 -5953.531} C_VEL
LIN {X 0,Y 503.766,Z 622.216,A -85,B 0,C 180,E1 -5955.164,E2 -5955.164} C_VEL
LIN {X 0,Y 504.291,Z 611.347,A -85,B 0,C 180,E1 -5956.601,E2 -5956.601} C_VEL
LIN {X 0,Y 505.035,Z 598.604,A -85,B 0,C 180,E1 -5958.037,E2 -5958.037} C_VEL
LIN {X 0,Y 505.879,Z 585.552,A -85,B 0,C 180,E1 -5959.283,E2 -5959.283} C_VEL
LIN {X 0,Y 506.685,Z 571.702,A -85,B 0,C 180,E1 -5960.396,E2 -5960.396} C_VEL
LIN {X 0,Y 507.453,Z 558.053,A -85,B 0,C 180,E1 -5961.311,E2 -5961.311} C_VEL
LIN {X 0,Y 508.224,Z 542.005,A -85,B 0,C 180,E1 -5962.191,E2 -5962.191} C_VEL
LIN {X 0,Y 508.88,Z 525.953,A -85,B 0,C 180,E1 -5962.885,E2 -5962.885} C_VEL
LIN {X 0,Y 509.173,Z 511.91,A -85,B 0,C 180,E1 -5963.363,E2 -5963.363} C_VEL
LIN {X 0,Y 503.007,Z 497.016,A -85,B 0,C 180,E1 -5964.041,E2 -5964.041} C_VEL
LIN {X 0,Y 502.856,Z 496.162,A -85,B 0,C 180,E1 -5964.075,E2 -5964.075} C_VEL
LIN {X 0,Y 502.868,Z 496.159,A -85,B 0,C 180,E1 -5966.566,E2 -5966.566} C_VEL
LIN {X 0,Y 502.828,Z 496.164,A -85,B 0,C 180,E1 -5969.288,E2 -5969.288} C_VEL
LIN {X 0,Y 502.787,Z 496.17,A -85,B 0,C 180,E1 -5972.085,E2 -5972.085} C_VEL
LIN {X 0,Y 502.813,Z 496.166,A -85,B 0,C 180,E1 -5974.965,E2 -5974.965} C_VEL
LIN {X 0,Y 502.799,Z 496.167,A -85,B 0,C 180,E1 -5977.954,E2 -5977.954} C_VEL
LIN {X 0,Y 502.824,Z 496.163,A -85,B 0,C 180,E1 -5981.066,E2 -5981.066} C_VEL
LIN {X 0,Y 502.791,Z 496.171,A -85,B 0,C 180,E1 -5984.53,E2 -5984.53} C_VEL
LIN {X 0,Y 502.803,Z 496.167,A -85,B 0,C 180,E1 -5987.861,E2 -5987.861} C_VEL
LIN {X 0,Y 502.792,Z 496.167,A -85,B 0,C 180,E1 -5988.175,E2 -5988.175} C_VEL
LIN {X 0,Y 502.13,Z 496.253,A -85,B 0,C 180,E1 -5988.843,E2 -5988.843} C_VEL
LIN {X 0,Y 499.287,Z 496.606,A -85,B 0,C 180,E1 -5989.93,E2 -5989.93} C_VEL
LIN {X 0,Y 496.874,Z 496.906,A -85,B 0,C 180,E1 -5990.805,E2 -5990.805} C_VEL
LIN {X 0,Y 495.825,Z 497.037,A -85,B 0,C 180,E1 -5991.48,E2 -5991.48} C_VEL
LIN {X 0,Y 495.733,Z 497.046,A -85,B 0,C 180,E1 -5991.709,E2 -5991.709} C_VEL
LIN {X 0,Y 495.754,Z 497.049,A -85,B 0,C 180,E1 -5994.462,E2 -5994.462} C_VEL
LIN {X 0,Y 495.773,Z 497.046,A -85,B 0,C 180,E1 -5997.406,E2 -5997.406} C_VEL
LIN {X 0,Y 495.772,Z 497.047,A -85,B 0,C 180,E1 -6000.253,E2 -6000.253} C_VEL
LIN {X 0,Y 495.83,Z 497.039,A -85,B 0,C 180,E1 -6003.251,E2 -6003.251} C_VEL
LIN {X 0,Y 495.909,Z 497.114,A -85,B 0,C 180,E1 -6005.364,E2 -6005.364} C_VEL
LIN {X 0,Y 495.86,Z 502.637,A -85,B 0,C 180,E1 -6008.376,E2 -6008.376} C_VEL
LIN {X 0,Y 495.831,Z 507.267,A -85,B 0,C 180,E1 -6010.973,E2 -6010.973} C_VEL
LIN {X 0,Y 495.737,Z 511.688,A -85,B 0,C 180,E1 -6013.528,E2 -6013.528} C_VEL
LIN {X 0,Y 495.679,Z 515.976,A -85,B 0,C 180,E1 -6016.052,E2 -6016.052} C_VEL
LIN {X 0,Y 495.675,Z 520.143,A -85,B 0,C 180,E1 -6018.55,E2 -6018.55} C_VEL
LIN {X 0,Y 495.545,Z 523.116,A -85,B 0,C 180,E1 -6020.352,E2 -6020.352} C_VEL
LIN {X 0,Y 498.357,Z 531.035,A -85,B 0,C 180,E1 -6020.636,E2 -6020.636} C_VEL
LIN {X 0,Y 503.061,Z 546.448,A -85,B 0,C 180,E1 -6021.23,E2 -6021.23} C_VEL
LIN {X 0,Y 502.551,Z 562.568,A -85,B 0,C 180,E1 -6021.732,E2 -6021.732} C_VEL
LIN {X 0,Y 501.881,Z 578.74,A -85,B 0,C 180,E1 -6022.405,E2 -6022.405} C_VEL
LIN {X 0,Y 501.163,Z 593.049,A -85,B 0,C 180,E1 -6023.153,E2 -6023.153} C_VEL
LIN {X 0,Y 500.249,Z 608.56,A -85,B 0,C 180,E1 -6024.153,E2 -6024.153} C_VEL
LIN {X 0,Y 499.333,Z 622.644,A -85,B 0,C 180,E1 -6025.256,E2 -6025.256} C_VEL
LIN {X 0,Y 498.402,Z 636.586,A -85,B 0,C 180,E1 -6026.563,E2 -6026.563} C_VEL
LIN {X 0,Y 497.667,Z 647.497,A -85,B 0,C 180,E1 -6027.774,E2 -6027.774} C_VEL
LIN {X 0,Y 497.04,Z 657.041,A -85,B 0,C 180,E1 -6028.986,E2 -6028.986} C_VEL
LIN {X 0,Y 496.363,Z 666.818,A -85,B 0,C 180,E1 -6030.405,E2 -6030.405} C_VEL
LIN {X 0,Y 495.945,Z 676.463,A -85,B 0,C 180,E1 -6032.029,E2 -6032.029} C_VEL
LIN {X 0,Y 495.536,Z 684.492,A -85,B 0,C 180,E1 -6033.658,E2 -6033.658} C_VEL
LIN {X 0,Y 495.284,Z 691.237,A -85,B 0,C 180,E1 -6035.291,E2 -6035.291} C_VEL
LIN {X 0,Y 495.205,Z 695.67,A -85,B 0,C 180,E1 -6036.56,E2 -6036.56} C_VEL
LIN {X 0,Y 495.091,Z 700.27,A -85,B 0,C 180,E1 -6038.16,E2 -6038.16} C_VEL
LIN {X 0,Y 495.002,Z 702.323,A -85,B 0,C 180,E1 -6038.984,E2 -6038.984} C_VEL
LIN {X 0,Y 494.945,Z 705.479,A -85,B 0,C 180,E1 -6040.636,E2 -6040.636} C_VEL
LIN {X 0,Y 494.917,Z 707.603,A -85,B 0,C 180,E1 -6042.297,E2 -6042.297} C_VEL
LIN {X 0,Y 494.897,Z 708.729,A -85,B 0,C 180,E1 -6043.969,E2 -6043.969} C_VEL
LIN {X 0,Y 494.894,Z 709,A -85,B 0,C 180,E1 -6045.055,E2 -6045.055} C_VEL
LIN {X 0,Y 494.849,Z 708.616,A -85,B 0,C 180,E1 -6046.501,E2 -6046.501} C_VEL
LIN {X 0,Y 494.882,Z 707.188,A -85,B 0,C 180,E1 -6048.205,E2 -6048.205} C_VEL
LIN {X 0,Y 494.971,Z 703.675,A -85,B 0,C 180,E1 -6050.425,E2 -6050.425} C_VEL
LIN {X 0,Y 495.075,Z 699.854,A -85,B 0,C 180,E1 -6052.097,E2 -6052.097} C_VEL
LIN {X 0,Y 495.223,Z 694.664,A -85,B 0,C 180,E1 -6053.856,E2 -6053.856} C_VEL
LIN {X 0,Y 495.43,Z 687.958,A -85,B 0,C 180,E1 -6055.635,E2 -6055.635} C_VEL
LIN {X 0,Y 495.745,Z 680.797,A -85,B 0,C 180,E1 -6057.205,E2 -6057.205} C_VEL
LIN {X 0,Y 496.145,Z 672.266,A -85,B 0,C 180,E1 -6058.79,E2 -6058.79} C_VEL
LIN {X 0,Y 496.708,Z 662.528,A -85,B 0,C 180,E1 -6060.333,E2 -6060.333} C_VEL
LIN {X 0,Y 497.44,Z 651.361,A -85,B 0,C 180,E1 -6061.855,E2 -6061.855} C_VEL
LIN {X 0,Y 498.217,Z 639.205,A -85,B 0,C 180,E1 -6063.255,E2 -6063.255} C_VEL
LIN {X 0,Y 498.998,Z 627.453,A -85,B 0,C 180,E1 -6064.41,E2 -6064.41} C_VEL
LIN {X 0,Y 499.897,Z 614.496,A -85,B 0,C 180,E1 -6065.497,E2 -6065.497} C_VEL
LIN {X 0,Y 500.696,Z 600.838,A -85,B 0,C 180,E1 -6066.467,E2 -6066.467} C_VEL
LIN {X 0,Y 501.519,Z 585.303,A -85,B 0,C 180,E1 -6067.368,E2 -6067.368} C_VEL
LIN {X 0,Y 502.249,Z 570.092,A -85,B 0,C 180,E1 -6068.071,E2 -6068.071} C_VEL
LIN {X 0,Y 502.841,Z 553.682,A -85,B 0,C 180,E1 -6068.657,E2 -6068.657} C_VEL
LIN {X 0,Y 503.065,Z 546.445,A -85,B 0,C 180,E1 -6068.862,E2 -6068.862} C_VEL
LIN {X 0,Y 498.445,Z 531.342,A -85,B 0,C 180,E1 -6069.446,E2 -6069.446} C_VEL
LIN {X 0,Y 495.443,Z 523.291,A -85,B 0,C 180,E1 -6069.74,E2 -6069.74} C_VEL
LIN {X 0,Y 495.59,Z 518.744,A -85,B 0,C 180,E1 -6072.488,E2 -6072.488} C_VEL
LIN {X 0,Y 495.694,Z 514.256,A -85,B 0,C 180,E1 -6075.144,E2 -6075.144} C_VEL
LIN {X 0,Y 495.81,Z 509.043,A -85,B 0,C 180,E1 -6078.224,E2 -6078.224} C_VEL
LIN {X 0,Y 495.826,Z 503.662,A -85,B 0,C 180,E1 -6081.221,E2 -6081.221} C_VEL
LIN {X 0,Y 495.92,Z 497.662,A -85,B 0,C 180,E1 -6084.476,E2 -6084.476} C_VEL
LIN {X 0,Y 495.803,Z 497.042,A -85,B 0,C 180,E1 -6084.923,E2 -6084.923} C_VEL
LIN {X 0,Y 495.762,Z 497.047,A -85,B 0,C 180,E1 -6087.405,E2 -6087.405} C_VEL
LIN {X 0,Y 495.774,Z 497.045,A -85,B 0,C 180,E1 -6090.254,E2 -6090.254} C_VEL
LIN {X 0,Y 495.825,Z 497.037,A -85,B 0,C 180,E1 -6093.247,E2 -6093.247} C_VEL
LIN {X 0,Y 495.752,Z 497.046,A -85,B 0,C 180,E1 -6095.725,E2 -6095.725} C_VEL
LIN {X 0,Y 495.752,Z 497.046,A -85,B 0,C 180,E1 -6098.371,E2 -6098.371} C_VEL
LIN {X 0,Y 495.776,Z 497.041,A -85,B 0,C 180,E1 -6100.971,E2 -6100.971} C_VEL
LIN {X 0,Y 495.771,Z 497.04,A -85,B 0,C 180,E1 -6103.529,E2 -6103.529} C_VEL
LIN {X 0,Y 495.785,Z 497.039,A -85,B 0,C 180,E1 -6106.055,E2 -6106.055} C_VEL
LIN {X 0,Y 495.859,Z 497.031,A -85,B 0,C 180,E1 -6108.555,E2 -6108.555} C_VEL
LIN {X 0,Y 495.863,Z 497.028,A -85,B 0,C 180,E1 -6111.852,E2 -6111.852} C_VEL
LIN {X 0,Y 495.908,Z 497.024,A -85,B 0,C 180,E1 -6114.306,E2 -6114.306} C_VEL
LIN {X 0,Y 495.986,Z 497.016,A -85,B 0,C 180,E1 -6117.563,E2 -6117.563} C_VEL
LIN {X 0,Y 495.987,Z 497.016,A -85,B 0,C 180,E1 -6120,E2 -6120} C_VEL
LIN {X 0,Y 495.985,Z 497.015,A -85,B 0,C 180,E1 -6122.436,E2 -6122.436} C_VEL
LIN {X 0,Y 495.887,Z 497.023,A -85,B 0,C 180,E1 -6125.693,E2 -6125.693} C_VEL
LIN {X 0,Y 495.862,Z 497.028,A -85,B 0,C 180,E1 -6128.148,E2 -6128.148} C_VEL
LIN {X 0,Y 495.864,Z 497.032,A -85,B 0,C 180,E1 -6131.445,E2 -6131.445} C_VEL
LIN {X 0,Y 495.778,Z 497.04,A -85,B 0,C 180,E1 -6134.783,E2 -6134.783} C_VEL
LIN {X 0,Y 495.776,Z 497.023,A -85,B 0,C 180,E1 -6137.319,E2 -6137.319} C_VEL
LIN {X 0,Y 495.767,Z 497.042,A -85,B 0,C 180,E1 -6139.89,E2 -6139.89} C_VEL
LIN {X 0,Y 495.753,Z 497.039,A -85,B 0,C 180,E1 -6142.863,E2 -6142.863} C_VEL
LIN {X 0,Y 495.789,Z 497.034,A -85,B 0,C 180,E1 -6146.068,E2 -6146.068} C_VEL
LIN {X 0,Y 495.769,Z 497.043,A -85,B 0,C 180,E1 -6148.815,E2 -6148.815} C_VEL
LIN {X 0,Y 495.749,Z 497.047,A -85,B 0,C 180,E1 -6151.727,E2 -6151.727} C_VEL
LIN {X 0,Y 495.767,Z 497.045,A -85,B 0,C 180,E1 -6154.696,E2 -6154.696} C_VEL
LIN {X 0,Y 495.725,Z 497.048,A -85,B 0,C 180,E1 -6157.562,E2 -6157.562} C_VEL
LIN {X 0,Y 495.777,Z 497.04,A -85,B 0,C 180,E1 -6160.698,E2 -6160.698} C_VEL
LIN {X 0,Y 495.725,Z 497.049,A -85,B 0,C 180,E1 -6163.696,E2 -6163.696} C_VEL
LIN {X 0,Y 495.741,Z 497.061,A -85,B 0,C 180,E1 -6164.359,E2 -6164.359} C_VEL
LIN {X 0,Y 497.922,Z 506.731,A -85,B 0,C 180,E1 -6167.353,E2 -6167.353} C_VEL
LIN {X 0,Y 499.368,Z 513.973,A -85,B 0,C 180,E1 -6169.462,E2 -6169.462} C_VEL
LIN {X 0,Y 499.385,Z 520.531,A -85,B 0,C 180,E1 -6171.227,E2 -6171.227} C_VEL
LIN {X 0,Y 498.912,Z 532.08,A -85,B 0,C 180,E1 -6174.227,E2 -6174.227} C_VEL
LIN {X 0,Y 498.361,Z 545.588,A -85,B 0,C 180,E1 -6177.598,E2 -6177.598} C_VEL
LIN {X 0,Y 497.966,Z 557.223,A -85,B 0,C 180,E1 -6180.4,E2 -6180.4} C_VEL
LIN {X 0,Y 497.48,Z 568.203,A -85,B 0,C 180,E1 -6183.125,E2 -6183.125} C_VEL
LIN {X 0,Y 497.096,Z 577.272,A -85,B 0,C 180,E1 -6185.32,E2 -6185.32} C_VEL
LIN {X 0,Y 503.105,Z 598.865,A -85,B 0,C 180,E1 -6186.019,E2 -6186.019} C_VEL
LIN {X 0,Y 502.742,Z 615.284,A -85,B 0,C 180,E1 -6186.462,E2 -6186.462} C_VEL
LIN {X 0,Y 502.083,Z 632.141,A -85,B 0,C 180,E1 -6187.09,E2 -6187.09} C_VEL
LIN {X 0,Y 501.299,Z 648.206,A -85,B 0,C 180,E1 -6187.874,E2 -6187.874} C_VEL
LIN {X 0,Y 500.383,Z 663.474,A -85,B 0,C 180,E1 -6188.799,E2 -6188.799} C_VEL
LIN {X 0,Y 499.589,Z 677.625,A -85,B 0,C 180,E1 -6189.84,E2 -6189.84} C_VEL
LIN {X 0,Y 498.763,Z 689.962,A -85,B 0,C 180,E1 -6190.902,E2 -6190.902} C_VEL
LIN {X 0,Y 497.979,Z 702.026,A -85,B 0,C 180,E1 -6192.125,E2 -6192.125} C_VEL
LIN {X 0,Y 497.251,Z 714.268,A -85,B 0,C 180,E1 -6193.581,E2 -6193.581} C_VEL
LIN {X 0,Y 496.638,Z 724.706,A -85,B 0,C 180,E1 -6195.034,E2 -6195.034} C_VEL
LIN {X 0,Y 496.036,Z 734.82,A -85,B 0,C 180,E1 -6196.69,E2 -6196.69} C_VEL
LIN {X 0,Y 495.753,Z 742.413,A -85,B 0,C 180,E1 -6198.165,E2 -6198.165} C_VEL
LIN {X 0,Y 495.383,Z 749.494,A -85,B 0,C 180,E1 -6199.786,E2 -6199.786} C_VEL
LIN {X 0,Y 495.207,Z 755.469,A -85,B 0,C 180,E1 -6201.431,E2 -6201.431} C_VEL
LIN {X 0,Y 495.1,Z 761.251,A -85,B 0,C 180,E1 -6203.48,E2 -6203.48} C_VEL
LIN {X 0,Y 494.983,Z 764.637,A -85,B 0,C 180,E1 -6205.114,E2 -6205.114} C_VEL
LIN {X 0,Y 495.022,Z 767.091,A -85,B 0,C 180,E1 -6206.745,E2 -6206.745} C_VEL
LIN {X 0,Y 494.956,Z 768.479,A -85,B 0,C 180,E1 -6208.374,E2 -6208.374} C_VEL
LIN {X 0,Y 494.893,Z 769,A -85,B 0,C 180,E1 -6210.001,E2 -6210.001} C_VEL
LIN {X 0,Y 494.957,Z 768.478,A -85,B 0,C 180,E1 -6211.628,E2 -6211.628} C_VEL
LIN {X 0,Y 495.023,Z 767.088,A -85,B 0,C 180,E1 -6213.256,E2 -6213.256} C_VEL
LIN {X 0,Y 494.984,Z 764.633,A -85,B 0,C 180,E1 -6214.888,E2 -6214.888} C_VEL
LIN {X 0,Y 495.102,Z 761.249,A -85,B 0,C 180,E1 -6216.521,E2 -6216.521} C_VEL
LIN {X 0,Y 495.208,Z 755.465,A -85,B 0,C 180,E1 -6218.571,E2 -6218.571} C_VEL
LIN {X 0,Y 495.469,Z 747.853,A -85,B 0,C 180,E1 -6220.627,E2 -6220.627} C_VEL
LIN {X 0,Y 495.853,Z 739.251,A -85,B 0,C 180,E1 -6222.484,E2 -6222.484} C_VEL
LIN {X 0,Y 496.31,Z 729.973,A -85,B 0,C 180,E1 -6224.139,E2 -6224.139} C_VEL
LIN {X 0,Y 496.858,Z 720.416,A -85,B 0,C 180,E1 -6225.591,E2 -6225.591} C_VEL
LIN {X 0,Y 497.537,Z 709.277,A -85,B 0,C 180,E1 -6227.045,E2 -6227.045} C_VEL
LIN {X 0,Y 498.292,Z 697.133,A -85,B 0,C 180,E1 -6228.397,E2 -6228.397} C_VEL
LIN {X 0,Y 499.177,Z 683.943,A -85,B 0,C 180,E1 -6229.635,E2 -6229.635} C_VEL
LIN {X 0,Y 499.985,Z 670.837,A -85,B 0,C 180,E1 -6230.682,E2 -6230.682} C_VEL
LIN {X 0,Y 500.886,Z 655.704,A -85,B 0,C 180,E1 -6231.694,E2 -6231.694} C_VEL
LIN {X 0,Y 501.73,Z 640.232,A -85,B 0,C 180,E1 -6232.537,E2 -6232.537} C_VEL
LIN {X 0,Y 502.385,Z 625.179,A -85,B 0,C 180,E1 -6233.189,E2 -6233.189} C_VEL
LIN {X 0,Y 502.928,Z 608.608,A -85,B 0,C 180,E1 -6233.735,E2 -6233.735} C_VEL
LIN {X 0,Y 503.074,Z 598.761,A -85,B 0,C 180,E1 -6233.985,E2 -6233.985} C_VEL
LIN {X 0,Y 497.07,Z 577.077,A -85,B 0,C 180,E1 -6234.701,E2 -6234.701} C_VEL
LIN {X 0,Y 497.672,Z 564.562,A -85,B 0,C 180,E1 -6237.777,E2 -6237.777} C_VEL
LIN {X 0,Y 497.992,Z 556.185,A -85,B 0,C 180,E1 -6239.833,E2 -6239.833} C_VEL
LIN {X 0,Y 498.217,Z 542.081,A -85,B 0,C 180,E1 -6242.895,E2 -6242.895} C_VEL
LIN {X 0,Y 498.355,Z 528.755,A -85,B 0,C 180,E1 -6245.821,E2 -6245.821} C_VEL
LIN {X 0,Y 498.432,Z 515.831,A -85,B 0,C 180,E1 -6248.75,E2 -6248.75} C_VEL
LIN {X 0,Y 498.336,Z 510.094,A -85,B 0,C 180,E1 -6250.117,E2 -6250.117} C_VEL
LIN {X 0,Y 496.372,Z 500.036,A -85,B 0,C 180,E1 -6252.814,E2 -6252.814} C_VEL
LIN {X 0,Y 495.748,Z 497.048,A -85,B 0,C 180,E1 -6253.758,E2 -6253.758} C_VEL
LIN {X 0,Y 495.736,Z 497.049,A -85,B 0,C 180,E1 -6256.305,E2 -6256.305} C_VEL
LIN {X 0,Y 495.768,Z 497.044,A -85,B 0,C 180,E1 -6259.301,E2 -6259.301} C_VEL
LIN {X 0,Y 495.732,Z 497.051,A -85,B 0,C 180,E1 -6262.439,E2 -6262.439} C_VEL
LIN {X 0,Y 495.785,Z 497.04,A -85,B 0,C 180,E1 -6265.458,E2 -6265.458} C_VEL
LIN {X 0,Y 495.757,Z 497.047,A -85,B 0,C 180,E1 -6268.364,E2 -6268.364} C_VEL
LIN {X 0,Y 495.789,Z 497.04,A -85,B 0,C 180,E1 -6271.507,E2 -6271.507} C_VEL
LIN {X 0,Y 495.793,Z 497.043,A -85,B 0,C 180,E1 -6273.933,E2 -6273.933} C_VEL
LIN {X 0,Y 495.809,Z 497.041,A -85,B 0,C 180,E1 -6275.745,E2 -6275.745} C_VEL
LIN {X 0,Y 499.568,Z 506.799,A -85,B 0,C 180,E1 -6276.161,E2 -6276.161} C_VEL
LIN {X 0,Y 502.618,Z 514.17,A -85,B 0,C 180,E1 -6276.518,E2 -6276.518} C_VEL
LIN {X 0,Y 502.093,Z 530.512,A -85,B 0,C 180,E1 -6277.089,E2 -6277.089} C_VEL
LIN {X 0,Y 501.372,Z 546.839,A -85,B 0,C 180,E1 -6277.839,E2 -6277.839} C_VEL
LIN {X 0,Y 500.581,Z 561.79,A -85,B 0,C 180,E1 -6278.699,E2 -6278.699} C_VEL
LIN {X 0,Y 499.787,Z 576.511,A -85,B 0,C 180,E1 -6279.741,E2 -6279.741} C_VEL
LIN {X 0,Y 498.878,Z 590.986,A -85,B 0,C 180,E1 -6280.983,E2 -6280.983} C_VEL
LIN {X 0,Y 497.966,Z 604.15,A -85,B 0,C 180,E1 -6282.336,E2 -6282.336} C_VEL
LIN {X 0,Y 497.179,Z 616.22,A -85,B 0,C 180,E1 -6283.815,E2 -6283.815} C_VEL
LIN {X 0,Y 496.557,Z 626.039,A -85,B 0,C 180,E1 -6285.241,E2 -6285.241} C_VEL
LIN {X 0,Y 495.915,Z 636.831,A -85,B 0,C 180,E1 -6287.103,E2 -6287.103} C_VEL
LIN {X 0,Y 495.642,Z 644.019,A -85,B 0,C 180,E1 -6288.55,E2 -6288.55} C_VEL
LIN {X 0,Y 495.298,Z 650.932,A -85,B 0,C 180,E1 -6290.197,E2 -6290.197} C_VEL
LIN {X 0,Y 495.189,Z 656.597,A -85,B 0,C 180,E1 -6291.841,E2 -6291.841} C_VEL
LIN {X 0,Y 495.104,Z 661.266,A -85,B 0,C 180,E1 -6293.54,E2 -6293.54} C_VEL
LIN {X 0,Y 494.985,Z 664.569,A -85,B 0,C 180,E1 -6295.113,E2 -6295.113} C_VEL
LIN {X 0,Y 495.026,Z 667.016,A -85,B 0,C 180,E1 -6296.745,E2 -6296.745} C_VEL
LIN {X 0,Y 494.956,Z 668.489,A -85,B 0,C 180,E1 -6298.373,E2 -6298.373} C_VEL
LIN {X 0,Y 494.896,Z 668.997,A -85,B 0,C 180,E1 -6300,E2 -6300} C_VEL
LIN {X 0,Y 494.956,Z 668.529,A -85,B 0,C 180,E1 -6301.628,E2 -6301.628} C_VEL
LIN {X 0,Y 495.027,Z 667.114,A -85,B 0,C 180,E1 -6303.256,E2 -6303.256} C_VEL
LIN {X 0,Y 494.985,Z 664.729,A -85,B 0,C 180,E1 -6304.887,E2 -6304.887} C_VEL
LIN {X 0,Y 495.106,Z 661.063,A -85,B 0,C 180,E1 -6306.632,E2 -6306.632} C_VEL
LIN {X 0,Y 495.202,Z 655.578,A -85,B 0,C 180,E1 -6308.57,E2 -6308.57} C_VEL
LIN {X 0,Y 495.379,Z 649.675,A -85,B 0,C 180,E1 -6310.215,E2 -6310.215} C_VEL
LIN {X 0,Y 495.755,Z 641.886,A -85,B 0,C 180,E1 -6311.994,E2 -6311.994} C_VEL
LIN {X 0,Y 496.157,Z 632.741,A -85,B 0,C 180,E1 -6313.725,E2 -6313.725} C_VEL
LIN {X 0,Y 496.825,Z 622.401,A -85,B 0,C 180,E1 -6315.381,E2 -6315.381} C_VEL
LIN {X 0,Y 497.454,Z 611.673,A -85,B 0,C 180,E1 -6316.836,E2 -6316.836} C_VEL
LIN {X 0,Y 498.263,Z 598.954,A -85,B 0,C 180,E1 -6318.291,E2 -6318.291} C_VEL
LIN {X 0,Y 499.128,Z 586.078,A -85,B 0,C 180,E1 -6319.532,E2 -6319.532} C_VEL
LIN {X 0,Y 500.003,Z 571.887,A -85,B 0,C 180,E1 -6320.681,E2 -6320.681} C_VEL
LIN {X 0,Y 500.818,Z 558.344,A -85,B 0,C 180,E1 -6321.596,E2 -6321.596} C_VEL
LIN {X 0,Y 501.587,Z 543.103,A -85,B 0,C 180,E1 -6322.446,E2 -6322.446} C_VEL
LIN {X 0,Y 502.294,Z 526.602,A -85,B 0,C 180,E1 -6323.172,E2 -6323.172} C_VEL
LIN {X 0,Y 502.573,Z 513.837,A -85,B 0,C 180,E1 -6323.62,E2 -6323.62} C_VEL
LIN {X 0,Y 495.895,Z 497.621,A -85,B 0,C 180,E1 -6324.385,E2 -6324.385} C_VEL
LIN {X 0,Y 495.813,Z 497.04,A -85,B 0,C 180,E1 -6324.405,E2 -6324.405} C_VEL
LIN {X 0,Y 495.817,Z 497.038,A -85,B 0,C 180,E1 -6326.974,E2 -6326.974} C_VEL
LIN {X 0,Y 495.769,Z 497.046,A -85,B 0,C 180,E1 -6330.147,E2 -6330.147} C_VEL
LIN {X 0,Y 495.798,Z 497.043,A -85,B 0,C 180,E1 -6333.245,E2 -6333.245} C_VEL
LIN {X 0,Y 495.732,Z 497.051,A -85,B 0,C 180,E1 -6336.09,E2 -6336.09} C_VEL
LIN {X 0,Y 495.768,Z 497.045,A -85,B 0,C 180,E1 -6338.768,E2 -6338.768} C_VEL
LIN {X 0,Y 495.76,Z 497.046,A -85,B 0,C 180,E1 -6341.781,E2 -6341.781} C_VEL
LIN {X 0,Y 495.742,Z 497.045,A -85,B 0,C 180,E1 -6345.141,E2 -6345.141} C_VEL
LIN {X 0,Y 495.763,Z 497.042,A -85,B 0,C 180,E1 -6348.219,E2 -6348.219} C_VEL
LIN {X 0,Y 495.756,Z 497.045,A -85,B 0,C 180,E1 -6351.408,E2 -6351.408} C_VEL
LIN {X 0,Y 495.733,Z 497.046,A -85,B 0,C 180,E1 -6351.709,E2 -6351.709} C_VEL
LIN {X 0,Y 495.054,Z 497.132,A -85,B 0,C 180,E1 -6352.387,E2 -6352.387} C_VEL
LIN {X 0,Y 492.217,Z 497.488,A -85,B 0,C 180,E1 -6353.488,E2 -6353.488} C_VEL
LIN {X 0,Y 489.829,Z 497.786,A -85,B 0,C 180,E1 -6354.376,E2 -6354.376} C_VEL
LIN {X 0,Y 488.804,Z 497.911,A -85,B 0,C 180,E1 -6355.061,E2 -6355.061} C_VEL
LIN {X 0,Y 488.72,Z 497.921,A -85,B 0,C 180,E1 -6355.293,E2 -6355.293} C_VEL
LIN {X 0,Y 488.709,Z 497.925,A -85,B 0,C 180,E1 -6358.046,E2 -6358.046} C_VEL
LIN {X 0,Y 488.729,Z 497.922,A -85,B 0,C 180,E1 -6360.729,E2 -6360.729} C_VEL
LIN {X 0,Y 488.766,Z 497.917,A -85,B 0,C 180,E1 -6363.528,E2 -6363.528} C_VEL
LIN {X 0,Y 488.847,Z 498.013,A -85,B 0,C 180,E1 -6365.251,E2 -6365.251} C_VEL
LIN {X 0,Y 488.837,Z 503.121,A -85,B 0,C 180,E1 -6368.049,E2 -6368.049} C_VEL
LIN {X 0,Y 488.802,Z 507.81,A -85,B 0,C 180,E1 -6370.688,E2 -6370.688} C_VEL
LIN {X 0,Y 488.721,Z 512.306,A -85,B 0,C 180,E1 -6373.285,E2 -6373.285} C_VEL
LIN {X 0,Y 488.679,Z 516.657,A -85,B 0,C 180,E1 -6375.848,E2 -6375.848} C_VEL
LIN {X 0,Y 488.662,Z 520.862,A -85,B 0,C 180,E1 -6378.383,E2 -6378.383} C_VEL
LIN {X 0,Y 488.509,Z 523.524,A -85,B 0,C 180,E1 -6379.979,E2 -6379.979} C_VEL
LIN {X 0,Y 491.485,Z 531.674,A -85,B 0,C 180,E1 -6380.278,E2 -6380.278} C_VEL
LIN {X 0,Y 495.583,Z 544.501,A -85,B 0,C 180,E1 -6380.788,E2 -6380.788} C_VEL
LIN {X 0,Y 496.603,Z 548.274,A -85,B 0,C 180,E1 -6380.941,E2 -6380.941} C_VEL
LIN {X 0,Y 495.993,Z 564.639,A -85,B 0,C 180,E1 -6381.471,E2 -6381.471} C_VEL
LIN {X 0,Y 495.272,Z 580.358,A -85,B 0,C 180,E1 -6382.149,E2 -6382.149} C_VEL
LIN {X 0,Y 494.466,Z 595.242,A -85,B 0,C 180,E1 -6382.958,E2 -6382.958} C_VEL
LIN {X 0,Y 493.62,Z 609.094,A -85,B 0,C 180,E1 -6383.869,E2 -6383.869} C_VEL
LIN {X 0,Y 492.629,Z 623.163,A -85,B 0,C 180,E1 -6384.986,E2 -6384.986} C_VEL
LIN {X 0,Y 491.718,Z 636.083,A -85,B 0,C 180,E1 -6386.209,E2 -6386.209} C_VEL
LIN {X 0,Y 490.859,Z 648.035,A -85,B 0,C 180,E1 -6387.537,E2 -6387.537} C_VEL
LIN {X 0,Y 490.117,Z 659.083,A -85,B 0,C 180,E1 -6388.972,E2 -6388.972} C_VEL
LIN {X 0,Y 489.3,Z 669.811,A -85,B 0,C 180,E1 -6390.616,E2 -6390.616} C_VEL
LIN {X 0,Y 488.825,Z 678.749,A -85,B 0,C 180,E1 -6392.265,E2 -6392.265} C_VEL
LIN {X 0,Y 488.464,Z 685.431,A -85,B 0,C 180,E1 -6393.711,E2 -6393.711} C_VEL
LIN {X 0,Y 488.254,Z 690.518,A -85,B 0,C 180,E1 -6394.954,E2 -6394.954} C_VEL
LIN {X 0,Y 488.105,Z 696.208,A -85,B 0,C 180,E1 -6396.614,E2 -6396.614} C_VEL
LIN {X 0,Y 488.037,Z 699.778,A -85,B 0,C 180,E1 -6397.862,E2 -6397.862} C_VEL
LIN {X 0,Y 487.89,Z 702.777,A -85,B 0,C 180,E1 -6399.116,E2 -6399.116} C_VEL
LIN {X 0,Y 487.858,Z 705.773,A -85,B 0,C 180,E1 -6400.793,E2 -6400.793} C_VEL
LIN {X 0,Y 487.801,Z 707.778,A -85,B 0,C 180,E1 -6402.48,E2 -6402.48} C_VEL
LIN {X 0,Y 487.816,Z 708.785,A -85,B 0,C 180,E1 -6404.176,E2 -6404.176} C_VEL
LIN {X 0,Y 487.786,Z 708.99,A -85,B 0,C 180,E1 -6405.129,E2 -6405.129} C_VEL
LIN {X 0,Y 487.748,Z 708.473,A -85,B 0,C 180,E1 -6406.748,E2 -6406.748} C_VEL
LIN {X 0,Y 487.796,Z 706.878,A -85,B 0,C 180,E1 -6408.479,E2 -6408.479} C_VEL
LIN {X 0,Y 487.868,Z 704.2,A -85,B 0,C 180,E1 -6410.225,E2 -6410.225} C_VEL
LIN {X 0,Y 487.932,Z 701.458,A -85,B 0,C 180,E1 -6411.548,E2 -6411.548} C_VEL
LIN {X 0,Y 488.06,Z 696.666,A -85,B 0,C 180,E1 -6413.327,E2 -6413.327} C_VEL
LIN {X 0,Y 488.279,Z 691.253,A -85,B 0,C 180,E1 -6414.934,E2 -6414.934} C_VEL
LIN {X 0,Y 488.524,Z 684.985,A -85,B 0,C 180,E1 -6416.484,E2 -6416.484} C_VEL
LIN {X 0,Y 488.958,Z 676.31,A -85,B 0,C 180,E1 -6418.314,E2 -6418.314} C_VEL
LIN {X 0,Y 489.56,Z 667.029,A -85,B 0,C 180,E1 -6419.923,E2 -6419.923} C_VEL
LIN {X 0,Y 490.171,Z 657.718,A -85,B 0,C 180,E1 -6421.314,E2 -6421.314} C_VEL
LIN {X 0,Y 491.018,Z 646.37,A -85,B 0,C 180,E1 -6422.76,E2 -6422.76} C_VEL
LIN {X 0,Y 491.875,Z 633.647,A -85,B 0,C 180,E1 -6424.136,E2 -6424.136} C_VEL
LIN {X 0,Y 492.78,Z 621.13,A -85,B 0,C 180,E1 -6425.281,E2 -6425.281} C_VEL
LIN {X 0,Y 493.66,Z 607.526,A -85,B 0,C 180,E1 -6426.34,E2 -6426.34} C_VEL
LIN {X 0,Y 494.584,Z 593.077,A -85,B 0,C 180,E1 -6427.273,E2 -6427.273} C_VEL
LIN {X 0,Y 495.359,Z 578.376,A -85,B 0,C 180,E1 -6428.043,E2 -6428.043} C_VEL
LIN {X 0,Y 496.031,Z 562.998,A -85,B 0,C 180,E1 -6428.685,E2 -6428.685} C_VEL
LIN {X 0,Y 496.518,Z 547.838,A -85,B 0,C 180,E1 -6429.169,E2 -6429.169} C_VEL
LIN {X 0,Y 492.127,Z 533.559,A -85,B 0,C 180,E1 -6429.741,E2 -6429.741} C_VEL
LIN {X 0,Y 488.466,Z 523.842,A -85,B 0,C 180,E1 -6430.11,E2 -6430.11} C_VEL
LIN {X 0,Y 488.583,Z 519.273,A -85,B 0,C 180,E1 -6432.81,E2 -6432.81} C_VEL
LIN {X 0,Y 488.733,Z 513.932,A -85,B 0,C 180,E1 -6435.97,E2 -6435.97} C_VEL
LIN {X 0,Y 488.78,Z 509.423,A -85,B 0,C 180,E1 -6438.591,E2 -6438.591} C_VEL
LIN {X 0,Y 488.811,Z 505.313,A -85,B 0,C 180,E1 -6440.93,E2 -6440.93} C_VEL
LIN {X 0,Y 488.91,Z 499.938,A -85,B 0,C 180,E1 -6443.887,E2 -6443.887} C_VEL
LIN {X 0,Y 488.772,Z 497.918,A -85,B 0,C 180,E1 -6445.042,E2 -6445.042} C_VEL
LIN {X 0,Y 488.699,Z 497.929,A -85,B 0,C 180,E1 -6448.044,E2 -6448.044} C_VEL
LIN {X 0,Y 488.726,Z 497.923,A -85,B 0,C 180,E1 -6450.729,E2 -6450.729} C_VEL
LIN {X 0,Y 488.758,Z 497.918,A -85,B 0,C 180,E1 -6453.528,E2 -6453.528} C_VEL
LIN {X 0,Y 488.694,Z 497.927,A -85,B 0,C 180,E1 -6456.254,E2 -6456.254} C_VEL
LIN {X 0,Y 488.738,Z 497.921,A -85,B 0,C 180,E1 -6459.174,E2 -6459.174} C_VEL
LIN {X 0,Y 488.749,Z 497.918,A -85,B 0,C 180,E1 -6461.627,E2 -6461.627} C_VEL
LIN {X 0,Y 488.752,Z 497.917,A -85,B 0,C 180,E1 -6464.999,E2 -6464.999} C_VEL
LIN {X 0,Y 488.821,Z 497.909,A -85,B 0,C 180,E1 -6468.388,E2 -6468.388} C_VEL
LIN {X 0,Y 488.808,Z 497.906,A -85,B 0,C 180,E1 -6471.733,E2 -6471.733} C_VEL
LIN {X 0,Y 488.864,Z 497.902,A -85,B 0,C 180,E1 -6474.224,E2 -6474.224} C_VEL
LIN {X 0,Y 488.954,Z 497.892,A -85,B 0,C 180,E1 -6477.528,E2 -6477.528} C_VEL
LIN {X 0,Y 488.958,Z 497.891,A -85,B 0,C 180,E1 -6480,E2 -6480} C_VEL
LIN {X 0,Y 488.953,Z 497.89,A -85,B 0,C 180,E1 -6482.471,E2 -6482.471} C_VEL
LIN {X 0,Y 488.846,Z 497.9,A -85,B 0,C 180,E1 -6485.775,E2 -6485.775} C_VEL
LIN {X 0,Y 488.807,Z 497.907,A -85,B 0,C 180,E1 -6488.266,E2 -6488.266} C_VEL
LIN {X 0,Y 488.822,Z 497.906,A -85,B 0,C 180,E1 -6491.612,E2 -6491.612} C_VEL
LIN {X 0,Y 488.75,Z 497.915,A -85,B 0,C 180,E1 -6495,E2 -6495} C_VEL
LIN {X 0,Y 488.743,Z 497.901,A -85,B 0,C 180,E1 -6498.442,E2 -6498.442} C_VEL
LIN {X 0,Y 488.729,Z 497.923,A -85,B 0,C 180,E1 -6501.069,E2 -6501.069} C_VEL
LIN {X 0,Y 488.69,Z 497.91,A -85,B 0,C 180,E1 -6503.745,E2 -6503.745} C_VEL
LIN {X 0,Y 488.788,Z 497.912,A -85,B 0,C 180,E1 -6506.946,E2 -6506.946} C_VEL
LIN {X 0,Y 488.708,Z 497.924,A -85,B 0,C 180,E1 -6510.365,E2 -6510.365} C_VEL
